    "phi" := "phi" + "w0c_6_12_1" * SIN(1 * 0.4 * "x") + "w0d_6_12_1" * COS(1 * 0.4 * "x");
    "phi" := "phi" + "w0c_6_12_2" * SIN(2 * 0.4 * "x") + "w0d_6_12_2" * COS(2 * 0.4 * "x");
    "phi" := "phi" + "w0c_6_12_3" * SIN(3 * 0.4 * "x") + "w0d_6_12_3" * COS(3 * 0.4 * "x");
    "phi" := "phi" + "w0c_6_12_4" * SIN(4 * 0.4 * "x") + "w0d_6_12_4" * COS(4 * 0.4 * "x");
    "phi" := "phi" + "w0c_6_12_5" * SIN(5 * 0.4 * "x") + "w0d_6_12_5" * COS(5 * 0.4 * "x");
    "phi" := "phi" + "w0c_6_12_6" * SIN(6 * 0.4 * "x") + "w0d_6_12_6" * COS(6 * 0.4 * "x");
    "acc" := "acc" + "phi";
    "x" := "feat_13";
    "phi" := "w0b_6_13" * "x" / (1.0 + EXP(-"x"));
    "phi" := "phi" + "w0c_6_13_1" * SIN(1 * 0.4 * "x") + "w0d_6_13_1" * COS(1 * 0.4 * "x");
    "phi" := "phi" + "w0c_6_13_2" * SIN(2 * 0.4 * "x") + "w0d_6_13_2" * COS(2 * 0.4 * "x");
    "phi" := "phi" + "w0c_6_13_3" * SIN(3 * 0.4 * "x") + "w0d_6_13_3" * COS(3 * 0.4 * "x");
    "phi" := "phi" + "w0c_6_13_4" * SIN(4 * 0.4 * "x") + "w0d_6_13_4" * COS(4 * 0.4 * "x");
    "phi" := "phi" + "w0c_6_13_5" * SIN(5 * 0.4 * "x") + "w0d_6_13_5" * COS(5 * 0.4 * "x");
    "phi" := "phi" + "w0c_6_13_6" * SIN(6 * 0.4 * "x") + "w0d_6_13_6" * COS(6 * 0.4 * "x");
    "acc" := "acc" + "phi";
    "x" := "feat_14";
    "phi" := "w0b_6_14" * "x" / (1.0 + EXP(-"x"));
    "phi" := "phi" + "w0c_6_14_1" * SIN(1 * 0.4 * "x") + "w0d_6_14_1" * COS(1 * 0.4 * "x");
    "phi" := "phi" + "w0c_6_14_2" * SIN(2 * 0.4 * "x") + "w0d_6_14_2" * COS(2 * 0.4 * "x");
    "phi" := "phi" + "w0c_6_14_3" * SIN(3 * 0.4 * "x") + "w0d_6_14_3" * COS(3 * 0.4 * "x");
    "phi" := "phi" + "w0c_6_14_4" * SIN(4 * 0.4 * "x") + "w0d_6_14_4" * COS(4 * 0.4 * "x");
    "phi" := "phi" + "w0c_6_14_5" * SIN(5 * 0.4 * "x") + "w0d_6_14_5" * COS(5 * 0.4 * "x");
    "phi" := "phi" + "w0c_6_14_6" * SIN(6 * 0.4 * "x") + "w0d_6_14_6" * COS(6 * 0.4 * "x");
    "acc" := "acc" + "phi";
    "x" := "feat_15";
    "phi" := "w0b_6_15" * "x" / (1.0 + EXP(-"x"));
    "phi" := "phi" + "w0c_6_15_1" * SIN(1 * 0.4 * "x") + "w0d_6_15_1" * COS(1 * 0.4 * "x");
    "phi" := "phi" + "w0c_6_15_2" * SIN(2 * 0.4 * "x") + "w0d_6_15_2" * COS(2 * 0.4 * "x");
    "phi" := "phi" + "w0c_6_15_3" * SIN(3 * 0.4 * "x") + "w0d_6_15_3" * COS(3 * 0.4 * "x");
    "phi" := "phi" + "w0c_6_15_4" * SIN(4 * 0.4 * "x") + "w0d_6_15_4" * COS(4 * 0.4 * "x");
    "phi" := "phi" + "w0c_6_15_5" * SIN(5 * 0.4 * "x") + "w0d_6_15_5" * COS(5 * 0.4 * "x");
    "phi" := "phi" + "w0c_6_15_6" * SIN(6 * 0.4 * "x") + "w0d_6_15_6" * COS(6 * 0.4 * "x");
    "acc" := "acc" + "phi";
    "x" := "feat_16";
    "phi" := "w0b_6_16" * "x" / (1.0 + EXP(-"x"));
    "phi" := "phi" + "w0c_6_16_1" * SIN(1 * 0.4 * "x") + "w0d_6_16_1" * COS(1 * 0.4 * "x");
    "phi" := "phi" + "w0c_6_16_2" * SIN(2 * 0.4 * "x") + "w0d_6_16_2" * COS(2 * 0.4 * "x");
    "phi" := "phi" + "w0c_6_16_3" * SIN(3 * 0.4 * "x") + "w0d_6_16_3" * COS(3 * 0.4 * "x");
    "phi" := "phi" + "w0c_6_16_4" * SIN(4 * 0.4 * "x") + "w0d_6_16_4" * COS(4 * 0.4 * "x");
    "phi" := "phi" + "w0c_6_16_5" * SIN(5 * 0.4 * "x") + "w0d_6_16_5" * COS(5 * 0.4 * "x");
    "phi" := "phi" + "w0c_6_16_6" * SIN(6 * 0.4 * "x") + "w0d_6_16_6" * COS(6 * 0.4 * "x");
    "acc" := "acc" + "phi";
    "x" := "feat_17";
    "phi" := "w0b_6_17" * "x" / (1.0 + EXP(-"x"));
    "phi" := "phi" + "w0c_6_17_1" * SIN(1 * 0.4 * "x") + "w0d_6_17_1" * COS(1 * 0.4 * "x");
    "phi" := "phi" + "w0c_6_17_2" * SIN(2 * 0.4 * "x") + "w0d_6_17_2" * COS(2 * 0.4 * "x");
    "phi" := "phi" + "w0c_6_17_3" * SIN(3 * 0.4 * "x") + "w0d_6_17_3" * COS(3 * 0.4 * "x");
    "phi" := "phi" + "w0c_6_17_4" * SIN(4 * 0.4 * "x") + "w0d_6_17_4" * COS(4 * 0.4 * "x");
    "phi" := "phi" + "w0c_6_17_5" * SIN(5 * 0.4 * "x") + "w0d_6_17_5" * COS(5 * 0.4 * "x");
    "phi" := "phi" + "w0c_6_17_6" * SIN(6 * 0.4 * "x") + "w0d_6_17_6" * COS(6 * 0.4 * "x");
    "acc" := "acc" + "phi";
    "x" := "feat_18";
    "phi" := "w0b_6_18" * "x" / (1.0 + EXP(-"x"));
    "phi" := "phi" + "w0c_6_18_1" * SIN(1 * 0.4 * "x") + "w0d_6_18_1" * COS(1 * 0.4 * "x");
    "phi" := "phi" + "w0c_6_18_2" * SIN(2 * 0.4 * "x") + "w0d_6_18_2" * COS(2 * 0.4 * "x");
    "phi" := "phi" + "w0c_6_18_3" * SIN(3 * 0.4 * "x") + "w0d_6_18_3" * COS(3 * 0.4 * "x");
    "phi" := "phi" + "w0c_6_18_4" * SIN(4 * 0.4 * "x") + "w0d_6_18_4" * COS(4 * 0.4 * "x");
    "phi" := "phi" + "w0c_6_18_5" * SIN(5 * 0.4 * "x") + "w0d_6_18_5" * COS(5 * 0.4 * "x");
    "phi" := "phi" + "w0c_6_18_6" * SIN(6 * 0.4 * "x") + "w0d_6_18_6" * COS(6 * 0.4 * "x");
    "acc" := "acc" + "phi";
    "x" := "feat_19";
    "phi" := "w0b_6_19" * "x" / (1.0 + EXP(-"x"));
    "phi" := "phi" + "w0c_6_19_1" * SIN(1 * 0.4 * "x") + "w0d_6_19_1" * COS(1 * 0.4 * "x");
    "phi" := "phi" + "w0c_6_19_2" * SIN(2 * 0.4 * "x") + "w0d_6_19_2" * COS(2 * 0.4 * "x");
    "phi" := "phi" + "w0c_6_19_3" * SIN(3 * 0.4 * "x") + "w0d_6_19_3" * COS(3 * 0.4 * "x");
    "phi" := "phi" + "w0c_6_19_4" * SIN(4 * 0.4 * "x") + "w0d_6_19_4" * COS(4 * 0.4 * "x");
    "phi" := "phi" + "w0c_6_19_5" * SIN(5 * 0.4 * "x") + "w0d_6_19_5" * COS(5 * 0.4 * "x");
    "phi" := "phi" + "w0c_6_19_6" * SIN(6 * 0.4 * "x") + "w0d_6_19_6" * COS(6 * 0.4 * "x");
    "acc" := "acc" + "phi";
    "x" := "feat_20";
    "phi" := "w0b_6_20" * "x" / (1.0 + EXP(-"x"));
    "phi" := "phi" + "w0c_6_20_1" * SIN(1 * 0.4 * "x") + "w0d_6_20_1" * COS(1 * 0.4 * "x");
    "phi" := "phi" + "w0c_6_20_2" * SIN(2 * 0.4 * "x") + "w0d_6_20_2" * COS(2 * 0.4 * "x");
    "phi" := "phi" + "w0c_6_20_3" * SIN(3 * 0.4 * "x") + "w0d_6_20_3" * COS(3 * 0.4 * "x");
    "phi" := "phi" + "w0c_6_20_4" * SIN(4 * 0.4 * "x") + "w0d_6_20_4" * COS(4 * 0.4 * "x");
    "phi" := "phi" + "w0c_6_20_5" * SIN(5 * 0.4 * "x") + "w0d_6_20_5" * COS(5 * 0.4 * "x");
    "phi" := "phi" + "w0c_6_20_6" * SIN(6 * 0.4 * "x") + "w0d_6_20_6" * COS(6 * 0.4 * "x");
    "acc" := "acc" + "phi";
    "x" := "feat_21";
    "phi" := "w0b_6_21" * "x" / (1.0 + EXP(-"x"));
    "phi" := "phi" + "w0c_6_21_1" * SIN(1 * 0.4 * "x") + "w0d_6_21_1" * COS(1 * 0.4 * "x");
    "phi" := "phi" + "w0c_6_21_2" * SIN(2 * 0.4 * "x") + "w0d_6_21_2" * COS(2 * 0.4 * "x");
    "phi" := "phi" + "w0c_6_21_3" * SIN(3 * 0.4 * "x") + "w0d_6_21_3" * COS(3 * 0.4 * "x");
    "phi" := "phi" + "w0c_6_21_4" * SIN(4 * 0.4 * "x") + "w0d_6_21_4" * COS(4 * 0.4 * "x");
    "phi" := "phi" + "w0c_6_21_5" * SIN(5 * 0.4 * "x") + "w0d_6_21_5" * COS(5 * 0.4 * "x");
    "phi" := "phi" + "w0c_6_21_6" * SIN(6 * 0.4 * "x") + "w0d_6_21_6" * COS(6 * 0.4 * "x");
    "acc" := "acc" + "phi";
    "x" := "feat_22";
    "phi" := "w0b_6_22" * "x" / (1.0 + EXP(-"x"));
    "phi" := "phi" + "w0c_6_22_1" * SIN(1 * 0.4 * "x") + "w0d_6_22_1" * COS(1 * 0.4 * "x");
    "phi" := "phi" + "w0c_6_22_2" * SIN(2 * 0.4 * "x") + "w0d_6_22_2" * COS(2 * 0.4 * "x");
    "phi" := "phi" + "w0c_6_22_3" * SIN(3 * 0.4 * "x") + "w0d_6_22_3" * COS(3 * 0.4 * "x");
    "phi" := "phi" + "w0c_6_22_4" * SIN(4 * 0.4 * "x") + "w0d_6_22_4" * COS(4 * 0.4 * "x");
    "phi" := "phi" + "w0c_6_22_5" * SIN(5 * 0.4 * "x") + "w0d_6_22_5" * COS(5 * 0.4 * "x");
    "phi" := "phi" + "w0c_6_22_6" * SIN(6 * 0.4 * "x") + "w0d_6_22_6" * COS(6 * 0.4 * "x");
    "acc" := "acc" + "phi";
    "x" := "feat_23";
    "phi" := "w0b_6_23" * "x" / (1.0 + EXP(-"x"));
    "phi" := "phi" + "w0c_6_23_1" * SIN(1 * 0.4 * "x") + "w0d_6_23_1" * COS(1 * 0.4 * "x");
    "phi" := "phi" + "w0c_6_23_2" * SIN(2 * 0.4 * "x") + "w0d_6_23_2" * COS(2 * 0.4 * "x");
    "phi" := "phi" + "w0c_6_23_3" * SIN(3 * 0.4 * "x") + "w0d_6_23_3" * COS(3 * 0.4 * "x");
    "phi" := "phi" + "w0c_6_23_4" * SIN(4 * 0.4 * "x") + "w0d_6_23_4" * COS(4 * 0.4 * "x");
    "phi" := "phi" + "w0c_6_23_5" * SIN(5 * 0.4 * "x") + "w0d_6_23_5" * COS(5 * 0.4 * "x");
    "phi" := "phi" + "w0c_6_23_6" * SIN(6 * 0.4 * "x") + "w0d_6_23_6" * COS(6 * 0.4 * "x");
    "acc" := "acc" + "phi";
    "x" := "feat_24";
    "phi" := "w0b_6_24" * "x" / (1.0 + EXP(-"x"));
    "phi" := "phi" + "w0c_6_24_1" * SIN(1 * 0.4 * "x") + "w0d_6_24_1" * COS(1 * 0.4 * "x");
    "phi" := "phi" + "w0c_6_24_2" * SIN(2 * 0.4 * "x") + "w0d_6_24_2" * COS(2 * 0.4 * "x");
    "phi" := "phi" + "w0c_6_24_3" * SIN(3 * 0.4 * "x") + "w0d_6_24_3" * COS(3 * 0.4 * "x");
    "phi" := "phi" + "w0c_6_24_4" * SIN(4 * 0.4 * "x") + "w0d_6_24_4" * COS(4 * 0.4 * "x");
    "phi" := "phi" + "w0c_6_24_5" * SIN(5 * 0.4 * "x") + "w0d_6_24_5" * COS(5 * 0.4 * "x");
    "phi" := "phi" + "w0c_6_24_6" * SIN(6 * 0.4 * "x") + "w0d_6_24_6" * COS(6 * 0.4 * "x");
    "acc" := "acc" + "phi";
    "x" := "feat_25";
    "phi" := "w0b_6_25" * "x" / (1.0 + EXP(-"x"));
    "phi" := "phi" + "w0c_6_25_1" * SIN(1 * 0.4 * "x") + "w0d_6_25_1" * COS(1 * 0.4 * "x");
    "phi" := "phi" + "w0c_6_25_2" * SIN(2 * 0.4 * "x") + "w0d_6_25_2" * COS(2 * 0.4 * "x");
    "phi" := "phi" + "w0c_6_25_3" * SIN(3 * 0.4 * "x") + "w0d_6_25_3" * COS(3 * 0.4 * "x");
    "phi" := "phi" + "w0c_6_25_4" * SIN(4 * 0.4 * "x") + "w0d_6_25_4" * COS(4 * 0.4 * "x");
    "phi" := "phi" + "w0c_6_25_5" * SIN(5 * 0.4 * "x") + "w0d_6_25_5" * COS(5 * 0.4 * "x");
    "phi" := "phi" + "w0c_6_25_6" * SIN(6 * 0.4 * "x") + "w0d_6_25_6" * COS(6 * 0.4 * "x");
    "acc" := "acc" + "phi";
    "x" := "feat_26";
    "phi" := "w0b_6_26" * "x" / (1.0 + EXP(-"x"));
    "phi" := "phi" + "w0c_6_26_1" * SIN(1 * 0.4 * "x") + "w0d_6_26_1" * COS(1 * 0.4 * "x");
    "phi" := "phi" + "w0c_6_26_2" * SIN(2 * 0.4 * "x") + "w0d_6_26_2" * COS(2 * 0.4 * "x");
    "phi" := "phi" + "w0c_6_26_3" * SIN(3 * 0.4 * "x") + "w0d_6_26_3" * COS(3 * 0.4 * "x");
    "phi" := "phi" + "w0c_6_26_4" * SIN(4 * 0.4 * "x") + "w0d_6_26_4" * COS(4 * 0.4 * "x");
    "phi" := "phi" + "w0c_6_26_5" * SIN(5 * 0.4 * "x") + "w0d_6_26_5" * COS(5 * 0.4 * "x");
    "phi" := "phi" + "w0c_6_26_6" * SIN(6 * 0.4 * "x") + "w0d_6_26_6" * COS(6 * 0.4 * "x");
    "acc" := "acc" + "phi";
    "x" := "feat_27";
    "phi" := "w0b_6_27" * "x" / (1.0 + EXP(-"x"));
    "phi" := "phi" + "w0c_6_27_1" * SIN(1 * 0.4 * "x") + "w0d_6_27_1" * COS(1 * 0.4 * "x");
    "phi" := "phi" + "w0c_6_27_2" * SIN(2 * 0.4 * "x") + "w0d_6_27_2" * COS(2 * 0.4 * "x");
    "phi" := "phi" + "w0c_6_27_3" * SIN(3 * 0.4 * "x") + "w0d_6_27_3" * COS(3 * 0.4 * "x");
    "phi" := "phi" + "w0c_6_27_4" * SIN(4 * 0.4 * "x") + "w0d_6_27_4" * COS(4 * 0.4 * "x");
    "phi" := "phi" + "w0c_6_27_5" * SIN(5 * 0.4 * "x") + "w0d_6_27_5" * COS(5 * 0.4 * "x");
    "phi" := "phi" + "w0c_6_27_6" * SIN(6 * 0.4 * "x") + "w0d_6_27_6" * COS(6 * 0.4 * "x");
    "acc" := "acc" + "phi";
    "x" := "feat_28";
    "phi" := "w0b_6_28" * "x" / (1.0 + EXP(-"x"));
    "phi" := "phi" + "w0c_6_28_1" * SIN(1 * 0.4 * "x") + "w0d_6_28_1" * COS(1 * 0.4 * "x");
    "phi" := "phi" + "w0c_6_28_2" * SIN(2 * 0.4 * "x") + "w0d_6_28_2" * COS(2 * 0.4 * "x");
    "phi" := "phi" + "w0c_6_28_3" * SIN(3 * 0.4 * "x") + "w0d_6_28_3" * COS(3 * 0.4 * "x");
    "phi" := "phi" + "w0c_6_28_4" * SIN(4 * 0.4 * "x") + "w0d_6_28_4" * COS(4 * 0.4 * "x");
    "phi" := "phi" + "w0c_6_28_5" * SIN(5 * 0.4 * "x") + "w0d_6_28_5" * COS(5 * 0.4 * "x");
    "phi" := "phi" + "w0c_6_28_6" * SIN(6 * 0.4 * "x") + "w0d_6_28_6" * COS(6 * 0.4 * "x");
    "acc" := "acc" + "phi";
    "h1_6" := "acc" + "b0_6";
    "acc" := 0.0;
    "x" := "feat_1";
    "phi" := "w0b_7_1" * "x" / (1.0 + EXP(-"x"));
    "phi" := "phi" + "w0c_7_1_1" * SIN(1 * 0.4 * "x") + "w0d_7_1_1" * COS(1 * 0.4 * "x");
    "phi" := "phi" + "w0c_7_1_2" * SIN(2 * 0.4 * "x") + "w0d_7_1_2" * COS(2 * 0.4 * "x");
    "phi" := "phi" + "w0c_7_1_3" * SIN(3 * 0.4 * "x") + "w0d_7_1_3" * COS(3 * 0.4 * "x");
    "phi" := "phi" + "w0c_7_1_4" * SIN(4 * 0.4 * "x") + "w0d_7_1_4" * COS(4 * 0.4 * "x");
    "phi" := "phi" + "w0c_7_1_5" * SIN(5 * 0.4 * "x") + "w0d_7_1_5" * COS(5 * 0.4 * "x");
    "phi" := "phi" + "w0c_7_1_6" * SIN(6 * 0.4 * "x") + "w0d_7_1_6" * COS(6 * 0.4 * "x");
    "acc" := "acc" + "phi";
    "x" := "feat_2";
    "phi" := "w0b_7_2" * "x" / (1.0 + EXP(-"x"));
    "phi" := "phi" + "w0c_7_2_1" * SIN(1 * 0.4 * "x") + "w0d_7_2_1" * COS(1 * 0.4 * "x");
    "phi" := "phi" + "w0c_7_2_2" * SIN(2 * 0.4 * "x") + "w0d_7_2_2" * COS(2 * 0.4 * "x");
    "phi" := "phi" + "w0c_7_2_3" * SIN(3 * 0.4 * "x") + "w0d_7_2_3" * COS(3 * 0.4 * "x");
    "phi" := "phi" + "w0c_7_2_4" * SIN(4 * 0.4 * "x") + "w0d_7_2_4" * COS(4 * 0.4 * "x");
    "phi" := "phi" + "w0c_7_2_5" * SIN(5 * 0.4 * "x") + "w0d_7_2_5" * COS(5 * 0.4 * "x");
    "phi" := "phi" + "w0c_7_2_6" * SIN(6 * 0.4 * "x") + "w0d_7_2_6" * COS(6 * 0.4 * "x");
    "acc" := "acc" + "phi";
    "x" := "feat_3";
    "phi" := "w0b_7_3" * "x" / (1.0 + EXP(-"x"));
    "phi" := "phi" + "w0c_7_3_1" * SIN(1 * 0.4 * "x") + "w0d_7_3_1" * COS(1 * 0.4 * "x");
    "phi" := "phi" + "w0c_7_3_2" * SIN(2 * 0.4 * "x") + "w0d_7_3_2" * COS(2 * 0.4 * "x");
    "phi" := "phi" + "w0c_7_3_3" * SIN(3 * 0.4 * "x") + "w0d_7_3_3" * COS(3 * 0.4 * "x");
    "phi" := "phi" + "w0c_7_3_4" * SIN(4 * 0.4 * "x") + "w0d_7_3_4" * COS(4 * 0.4 * "x");
    "phi" := "phi" + "w0c_7_3_5" * SIN(5 * 0.4 * "x") + "w0d_7_3_5" * COS(5 * 0.4 * "x");
    "phi" := "phi" + "w0c_7_3_6" * SIN(6 * 0.4 * "x") + "w0d_7_3_6" * COS(6 * 0.4 * "x");
    "acc" := "acc" + "phi";
    "x" := "feat_4";
    "phi" := "w0b_7_4" * "x" / (1.0 + EXP(-"x"));
    "phi" := "phi" + "w0c_7_4_1" * SIN(1 * 0.4 * "x") + "w0d_7_4_1" * COS(1 * 0.4 * "x");
    "phi" := "phi" + "w0c_7_4_2" * SIN(2 * 0.4 * "x") + "w0d_7_4_2" * COS(2 * 0.4 * "x");
    "phi" := "phi" + "w0c_7_4_3" * SIN(3 * 0.4 * "x") + "w0d_7_4_3" * COS(3 * 0.4 * "x");
    "phi" := "phi" + "w0c_7_4_4" * SIN(4 * 0.4 * "x") + "w0d_7_4_4" * COS(4 * 0.4 * "x");
    "phi" := "phi" + "w0c_7_4_5" * SIN(5 * 0.4 * "x") + "w0d_7_4_5" * COS(5 * 0.4 * "x");
    "phi" := "phi" + "w0c_7_4_6" * SIN(6 * 0.4 * "x") + "w0d_7_4_6" * COS(6 * 0.4 * "x");
    "acc" := "acc" + "phi";
    "x" := "feat_5";
    "phi" := "w0b_7_5" * "x" / (1.0 + EXP(-"x"));
    "phi" := "phi" + "w0c_7_5_1" * SIN(1 * 0.4 * "x") + "w0d_7_5_1" * COS(1 * 0.4 * "x");
    "phi" := "phi" + "w0c_7_5_2" * SIN(2 * 0.4 * "x") + "w0d_7_5_2" * COS(2 * 0.4 * "x");
    "phi" := "phi" + "w0c_7_5_3" * SIN(3 * 0.4 * "x") + "w0d_7_5_3" * COS(3 * 0.4 * "x");
    "phi" := "phi" + "w0c_7_5_4" * SIN(4 * 0.4 * "x") + "w0d_7_5_4" * COS(4 * 0.4 * "x");
    "phi" := "phi" + "w0c_7_5_5" * SIN(5 * 0.4 * "x") + "w0d_7_5_5" * COS(5 * 0.4 * "x");
    "phi" := "phi" + "w0c_7_5_6" * SIN(6 * 0.4 * "x") + "w0d_7_5_6" * COS(6 * 0.4 * "x");
    "acc" := "acc" + "phi";
    "x" := "feat_6";
    "phi" := "w0b_7_6" * "x" / (1.0 + EXP(-"x"));
    "phi" := "phi" + "w0c_7_6_1" * SIN(1 * 0.4 * "x") + "w0d_7_6_1" * COS(1 * 0.4 * "x");
    "phi" := "phi" + "w0c_7_6_2" * SIN(2 * 0.4 * "x") + "w0d_7_6_2" * COS(2 * 0.4 * "x");
    "phi" := "phi" + "w0c_7_6_3" * SIN(3 * 0.4 * "x") + "w0d_7_6_3" * COS(3 * 0.4 * "x");
    "phi" := "phi" + "w0c_7_6_4" * SIN(4 * 0.4 * "x") + "w0d_7_6_4" * COS(4 * 0.4 * "x");
    "phi" := "phi" + "w0c_7_6_5" * SIN(5 * 0.4 * "x") + "w0d_7_6_5" * COS(5 * 0.4 * "x");
    "phi" := "phi" + "w0c_7_6_6" * SIN(6 * 0.4 * "x") + "w0d_7_6_6" * COS(6 * 0.4 * "x");
    "acc" := "acc" + "phi";
    "x" := "feat_7";
    "phi" := "w0b_7_7" * "x" / (1.0 + EXP(-"x"));
    "phi" := "phi" + "w0c_7_7_1" * SIN(1 * 0.4 * "x") + "w0d_7_7_1" * COS(1 * 0.4 * "x");
    "phi" := "phi" + "w0c_7_7_2" * SIN(2 * 0.4 * "x") + "w0d_7_7_2" * COS(2 * 0.4 * "x");
    "phi" := "phi" + "w0c_7_7_3" * SIN(3 * 0.4 * "x") + "w0d_7_7_3" * COS(3 * 0.4 * "x");
    "phi" := "phi" + "w0c_7_7_4" * SIN(4 * 0.4 * "x") + "w0d_7_7_4" * COS(4 * 0.4 * "x");
    "phi" := "phi" + "w0c_7_7_5" * SIN(5 * 0.4 * "x") + "w0d_7_7_5" * COS(5 * 0.4 * "x");
    "phi" := "phi" + "w0c_7_7_6" * SIN(6 * 0.4 * "x") + "w0d_7_7_6" * COS(6 * 0.4 * "x");
    "acc" := "acc" + "phi";
    "x" := "feat_8";
    "phi" := "w0b_7_8" * "x" / (1.0 + EXP(-"x"));
    "phi" := "phi" + "w0c_7_8_1" * SIN(1 * 0.4 * "x") + "w0d_7_8_1" * COS(1 * 0.4 * "x");
    "phi" := "phi" + "w0c_7_8_2" * SIN(2 * 0.4 * "x") + "w0d_7_8_2" * COS(2 * 0.4 * "x");
    "phi" := "phi" + "w0c_7_8_3" * SIN(3 * 0.4 * "x") + "w0d_7_8_3" * COS(3 * 0.4 * "x");
    "phi" := "phi" + "w0c_7_8_4" * SIN(4 * 0.4 * "x") + "w0d_7_8_4" * COS(4 * 0.4 * "x");
    "phi" := "phi" + "w0c_7_8_5" * SIN(5 * 0.4 * "x") + "w0d_7_8_5" * COS(5 * 0.4 * "x");
    "phi" := "phi" + "w0c_7_8_6" * SIN(6 * 0.4 * "x") + "w0d_7_8_6" * COS(6 * 0.4 * "x");
    "acc" := "acc" + "phi";
    "x" := "feat_9";
    "phi" := "w0b_7_9" * "x" / (1.0 + EXP(-"x"));
    "phi" := "phi" + "w0c_7_9_1" * SIN(1 * 0.4 * "x") + "w0d_7_9_1" * COS(1 * 0.4 * "x");
    "phi" := "phi" + "w0c_7_9_2" * SIN(2 * 0.4 * "x") + "w0d_7_9_2" * COS(2 * 0.4 * "x");
    "phi" := "phi" + "w0c_7_9_3" * SIN(3 * 0.4 * "x") + "w0d_7_9_3" * COS(3 * 0.4 * "x");
    "phi" := "phi" + "w0c_7_9_4" * SIN(4 * 0.4 * "x") + "w0d_7_9_4" * COS(4 * 0.4 * "x");
    "phi" := "phi" + "w0c_7_9_5" * SIN(5 * 0.4 * "x") + "w0d_7_9_5" * COS(5 * 0.4 * "x");
    "phi" := "phi" + "w0c_7_9_6" * SIN(6 * 0.4 * "x") + "w0d_7_9_6" * COS(6 * 0.4 * "x");
    "acc" := "acc" + "phi";
    "x" := "feat_10";
    "phi" := "w0b_7_10" * "x" / (1.0 + EXP(-"x"));
    "phi" := "phi" + "w0c_7_10_1" * SIN(1 * 0.4 * "x") + "w0d_7_10_1" * COS(1 * 0.4 * "x");
    "phi" := "phi" + "w0c_7_10_2" * SIN(2 * 0.4 * "x") + "w0d_7_10_2" * COS(2 * 0.4 * "x");
    "phi" := "phi" + "w0c_7_10_3" * SIN(3 * 0.4 * "x") + "w0d_7_10_3" * COS(3 * 0.4 * "x");
    "phi" := "phi" + "w0c_7_10_4" * SIN(4 * 0.4 * "x") + "w0d_7_10_4" * COS(4 * 0.4 * "x");
    "phi" := "phi" + "w0c_7_10_5" * SIN(5 * 0.4 * "x") + "w0d_7_10_5" * COS(5 * 0.4 * "x");
    "phi" := "phi" + "w0c_7_10_6" * SIN(6 * 0.4 * "x") + "w0d_7_10_6" * COS(6 * 0.4 * "x");
    "acc" := "acc" + "phi";
    "x" := "feat_11";
    "phi" := "w0b_7_11" * "x" / (1.0 + EXP(-"x"));
    "phi" := "phi" + "w0c_7_11_1" * SIN(1 * 0.4 * "x") + "w0d_7_11_1" * COS(1 * 0.4 * "x");
    "phi" := "phi" + "w0c_7_11_2" * SIN(2 * 0.4 * "x") + "w0d_7_11_2" * COS(2 * 0.4 * "x");
    "phi" := "phi" + "w0c_7_11_3" * SIN(3 * 0.4 * "x") + "w0d_7_11_3" * COS(3 * 0.4 * "x");
    "phi" := "phi" + "w0c_7_11_4" * SIN(4 * 0.4 * "x") + "w0d_7_11_4" * COS(4 * 0.4 * "x");
    "phi" := "phi" + "w0c_7_11_5" * SIN(5 * 0.4 * "x") + "w0d_7_11_5" * COS(5 * 0.4 * "x");
    "phi" := "phi" + "w0c_7_11_6" * SIN(6 * 0.4 * "x") + "w0d_7_11_6" * COS(6 * 0.4 * "x");
    "acc" := "acc" + "phi";
    "x" := "feat_12";
    "phi" := "w0b_7_12" * "x" / (1.0 + EXP(-"x"));
    "phi" := "phi" + "w0c_7_12_1" * SIN(1 * 0.4 * "x") + "w0d_7_12_1" * COS(1 * 0.4 * "x");
    "phi" := "phi" + "w0c_7_12_2" * SIN(2 * 0.4 * "x") + "w0d_7_12_2" * COS(2 * 0.4 * "x");
    "phi" := "phi" + "w0c_7_12_3" * SIN(3 * 0.4 * "x") + "w0d_7_12_3" * COS(3 * 0.4 * "x");
    "phi" := "phi" + "w0c_7_12_4" * SIN(4 * 0.4 * "x") + "w0d_7_12_4" * COS(4 * 0.4 * "x");
    "phi" := "phi" + "w0c_7_12_5" * SIN(5 * 0.4 * "x") + "w0d_7_12_5" * COS(5 * 0.4 * "x");
    "phi" := "phi" + "w0c_7_12_6" * SIN(6 * 0.4 * "x") + "w0d_7_12_6" * COS(6 * 0.4 * "x");
    "acc" := "acc" + "phi";
    "x" := "feat_13";
    "phi" := "w0b_7_13" * "x" / (1.0 + EXP(-"x"));
    "phi" := "phi" + "w0c_7_13_1" * SIN(1 * 0.4 * "x") + "w0d_7_13_1" * COS(1 * 0.4 * "x");
    "phi" := "phi" + "w0c_7_13_2" * SIN(2 * 0.4 * "x") + "w0d_7_13_2" * COS(2 * 0.4 * "x");
    "phi" := "phi" + "w0c_7_13_3" * SIN(3 * 0.4 * "x") + "w0d_7_13_3" * COS(3 * 0.4 * "x");
    "phi" := "phi" + "w0c_7_13_4" * SIN(4 * 0.4 * "x") + "w0d_7_13_4" * COS(4 * 0.4 * "x");
    "phi" := "phi" + "w0c_7_13_5" * SIN(5 * 0.4 * "x") + "w0d_7_13_5" * COS(5 * 0.4 * "x");
    "phi" := "phi" + "w0c_7_13_6" * SIN(6 * 0.4 * "x") + "w0d_7_13_6" * COS(6 * 0.4 * "x");
    "acc" := "acc" + "phi";
    "x" := "feat_14";
    "phi" := "w0b_7_14" * "x" / (1.0 + EXP(-"x"));
    "phi" := "phi" + "w0c_7_14_1" * SIN(1 * 0.4 * "x") + "w0d_7_14_1" * COS(1 * 0.4 * "x");
    "phi" := "phi" + "w0c_7_14_2" * SIN(2 * 0.4 * "x") + "w0d_7_14_2" * COS(2 * 0.4 * "x");
    "phi" := "phi" + "w0c_7_14_3" * SIN(3 * 0.4 * "x") + "w0d_7_14_3" * COS(3 * 0.4 * "x");
    "phi" := "phi" + "w0c_7_14_4" * SIN(4 * 0.4 * "x") + "w0d_7_14_4" * COS(4 * 0.4 * "x");
    "phi" := "phi" + "w0c_7_14_5" * SIN(5 * 0.4 * "x") + "w0d_7_14_5" * COS(5 * 0.4 * "x");
    "phi" := "phi" + "w0c_7_14_6" * SIN(6 * 0.4 * "x") + "w0d_7_14_6" * COS(6 * 0.4 * "x");
    "acc" := "acc" + "phi";
    "x" := "feat_15";
    "phi" := "w0b_7_15" * "x" / (1.0 + EXP(-"x"));
    "phi" := "phi" + "w0c_7_15_1" * SIN(1 * 0.4 * "x") + "w0d_7_15_1" * COS(1 * 0.4 * "x");
    "phi" := "phi" + "w0c_7_15_2" * SIN(2 * 0.4 * "x") + "w0d_7_15_2" * COS(2 * 0.4 * "x");
    "phi" := "phi" + "w0c_7_15_3" * SIN(3 * 0.4 * "x") + "w0d_7_15_3" * COS(3 * 0.4 * "x");
    "phi" := "phi" + "w0c_7_15_4" * SIN(4 * 0.4 * "x") + "w0d_7_15_4" * COS(4 * 0.4 * "x");
    "phi" := "phi" + "w0c_7_15_5" * SIN(5 * 0.4 * "x") + "w0d_7_15_5" * COS(5 * 0.4 * "x");
    "phi" := "phi" + "w0c_7_15_6" * SIN(6 * 0.4 * "x") + "w0d_7_15_6" * COS(6 * 0.4 * "x");
    "acc" := "acc" + "phi";
    "x" := "feat_16";
    "phi" := "w0b_7_16" * "x" / (1.0 + EXP(-"x"));
    "phi" := "phi" + "w0c_7_16_1" * SIN(1 * 0.4 * "x") + "w0d_7_16_1" * COS(1 * 0.4 * "x");
    "phi" := "phi" + "w0c_7_16_2" * SIN(2 * 0.4 * "x") + "w0d_7_16_2" * COS(2 * 0.4 * "x");
    "phi" := "phi" + "w0c_7_16_3" * SIN(3 * 0.4 * "x") + "w0d_7_16_3" * COS(3 * 0.4 * "x");
    "phi" := "phi" + "w0c_7_16_4" * SIN(4 * 0.4 * "x") + "w0d_7_16_4" * COS(4 * 0.4 * "x");
    "phi" := "phi" + "w0c_7_16_5" * SIN(5 * 0.4 * "x") + "w0d_7_16_5" * COS(5 * 0.4 * "x");
    "phi" := "phi" + "w0c_7_16_6" * SIN(6 * 0.4 * "x") + "w0d_7_16_6" * COS(6 * 0.4 * "x");
    "acc" := "acc" + "phi";
    "x" := "feat_17";
    "phi" := "w0b_7_17" * "x" / (1.0 + EXP(-"x"));
    "phi" := "phi" + "w0c_7_17_1" * SIN(1 * 0.4 * "x") + "w0d_7_17_1" * COS(1 * 0.4 * "x");
    "phi" := "phi" + "w0c_7_17_2" * SIN(2 * 0.4 * "x") + "w0d_7_17_2" * COS(2 * 0.4 * "x");
    "phi" := "phi" + "w0c_7_17_3" * SIN(3 * 0.4 * "x") + "w0d_7_17_3" * COS(3 * 0.4 * "x");
    "phi" := "phi" + "w0c_7_17_4" * SIN(4 * 0.4 * "x") + "w0d_7_17_4" * COS(4 * 0.4 * "x");
    "phi" := "phi" + "w0c_7_17_5" * SIN(5 * 0.4 * "x") + "w0d_7_17_5" * COS(5 * 0.4 * "x");
    "phi" := "phi" + "w0c_7_17_6" * SIN(6 * 0.4 * "x") + "w0d_7_17_6" * COS(6 * 0.4 * "x");
    "acc" := "acc" + "phi";
    "x" := "feat_18";
    "phi" := "w0b_7_18" * "x" / (1.0 + EXP(-"x"));
    "phi" := "phi" + "w0c_7_18_1" * SIN(1 * 0.4 * "x") + "w0d_7_18_1" * COS(1 * 0.4 * "x");
    "phi" := "phi" + "w0c_7_18_2" * SIN(2 * 0.4 * "x") + "w0d_7_18_2" * COS(2 * 0.4 * "x");
    "phi" := "phi" + "w0c_7_18_3" * SIN(3 * 0.4 * "x") + "w0d_7_18_3" * COS(3 * 0.4 * "x");
    "phi" := "phi" + "w0c_7_18_4" * SIN(4 * 0.4 * "x") + "w0d_7_18_4" * COS(4 * 0.4 * "x");
    "phi" := "phi" + "w0c_7_18_5" * SIN(5 * 0.4 * "x") + "w0d_7_18_5" * COS(5 * 0.4 * "x");
    "phi" := "phi" + "w0c_7_18_6" * SIN(6 * 0.4 * "x") + "w0d_7_18_6" * COS(6 * 0.4 * "x");
    "acc" := "acc" + "phi";
    "x" := "feat_19";
    "phi" := "w0b_7_19" * "x" / (1.0 + EXP(-"x"));
    "phi" := "phi" + "w0c_7_19_1" * SIN(1 * 0.4 * "x") + "w0d_7_19_1" * COS(1 * 0.4 * "x");
    "phi" := "phi" + "w0c_7_19_2" * SIN(2 * 0.4 * "x") + "w0d_7_19_2" * COS(2 * 0.4 * "x");
    "phi" := "phi" + "w0c_7_19_3" * SIN(3 * 0.4 * "x") + "w0d_7_19_3" * COS(3 * 0.4 * "x");
    "phi" := "phi" + "w0c_7_19_4" * SIN(4 * 0.4 * "x") + "w0d_7_19_4" * COS(4 * 0.4 * "x");
    "phi" := "phi" + "w0c_7_19_5" * SIN(5 * 0.4 * "x") + "w0d_7_19_5" * COS(5 * 0.4 * "x");
    "phi" := "phi" + "w0c_7_19_6" * SIN(6 * 0.4 * "x") + "w0d_7_19_6" * COS(6 * 0.4 * "x");
    "acc" := "acc" + "phi";
    "x" := "feat_20";
    "phi" := "w0b_7_20" * "x" / (1.0 + EXP(-"x"));
    "phi" := "phi" + "w0c_7_20_1" * SIN(1 * 0.4 * "x") + "w0d_7_20_1" * COS(1 * 0.4 * "x");
    "phi" := "phi" + "w0c_7_20_2" * SIN(2 * 0.4 * "x") + "w0d_7_20_2" * COS(2 * 0.4 * "x");
    "phi" := "phi" + "w0c_7_20_3" * SIN(3 * 0.4 * "x") + "w0d_7_20_3" * COS(3 * 0.4 * "x");
    "phi" := "phi" + "w0c_7_20_4" * SIN(4 * 0.4 * "x") + "w0d_7_20_4" * COS(4 * 0.4 * "x");
    "phi" := "phi" + "w0c_7_20_5" * SIN(5 * 0.4 * "x") + "w0d_7_20_5" * COS(5 * 0.4 * "x");
    "phi" := "phi" + "w0c_7_20_6" * SIN(6 * 0.4 * "x") + "w0d_7_20_6" * COS(6 * 0.4 * "x");
    "acc" := "acc" + "phi";
    "x" := "feat_21";
    "phi" := "w0b_7_21" * "x" / (1.0 + EXP(-"x"));
    "phi" := "phi" + "w0c_7_21_1" * SIN(1 * 0.4 * "x") + "w0d_7_21_1" * COS(1 * 0.4 * "x");
    "phi" := "phi" + "w0c_7_21_2" * SIN(2 * 0.4 * "x") + "w0d_7_21_2" * COS(2 * 0.4 * "x");
    "phi" := "phi" + "w0c_7_21_3" * SIN(3 * 0.4 * "x") + "w0d_7_21_3" * COS(3 * 0.4 * "x");
    "phi" := "phi" + "w0c_7_21_4" * SIN(4 * 0.4 * "x") + "w0d_7_21_4" * COS(4 * 0.4 * "x");
    "phi" := "phi" + "w0c_7_21_5" * SIN(5 * 0.4 * "x") + "w0d_7_21_5" * COS(5 * 0.4 * "x");
    "phi" := "phi" + "w0c_7_21_6" * SIN(6 * 0.4 * "x") + "w0d_7_21_6" * COS(6 * 0.4 * "x");
    "acc" := "acc" + "phi";
    "x" := "feat_22";
    "phi" := "w0b_7_22" * "x" / (1.0 + EXP(-"x"));
    "phi" := "phi" + "w0c_7_22_1" * SIN(1 * 0.4 * "x") + "w0d_7_22_1" * COS(1 * 0.4 * "x");
    "phi" := "phi" + "w0c_7_22_2" * SIN(2 * 0.4 * "x") + "w0d_7_22_2" * COS(2 * 0.4 * "x");
    "phi" := "phi" + "w0c_7_22_3" * SIN(3 * 0.4 * "x") + "w0d_7_22_3" * COS(3 * 0.4 * "x");
    "phi" := "phi" + "w0c_7_22_4" * SIN(4 * 0.4 * "x") + "w0d_7_22_4" * COS(4 * 0.4 * "x");
    "phi" := "phi" + "w0c_7_22_5" * SIN(5 * 0.4 * "x") + "w0d_7_22_5" * COS(5 * 0.4 * "x");
    "phi" := "phi" + "w0c_7_22_6" * SIN(6 * 0.4 * "x") + "w0d_7_22_6" * COS(6 * 0.4 * "x");
    "acc" := "acc" + "phi";
    "x" := "feat_23";
    "phi" := "w0b_7_23" * "x" / (1.0 + EXP(-"x"));
    "phi" := "phi" + "w0c_7_23_1" * SIN(1 * 0.4 * "x") + "w0d_7_23_1" * COS(1 * 0.4 * "x");
    "phi" := "phi" + "w0c_7_23_2" * SIN(2 * 0.4 * "x") + "w0d_7_23_2" * COS(2 * 0.4 * "x");
    "phi" := "phi" + "w0c_7_23_3" * SIN(3 * 0.4 * "x") + "w0d_7_23_3" * COS(3 * 0.4 * "x");
    "phi" := "phi" + "w0c_7_23_4" * SIN(4 * 0.4 * "x") + "w0d_7_23_4" * COS(4 * 0.4 * "x");
    "phi" := "phi" + "w0c_7_23_5" * SIN(5 * 0.4 * "x") + "w0d_7_23_5" * COS(5 * 0.4 * "x");
    "phi" := "phi" + "w0c_7_23_6" * SIN(6 * 0.4 * "x") + "w0d_7_23_6" * COS(6 * 0.4 * "x");
    "acc" := "acc" + "phi";
    "x" := "feat_24";
    "phi" := "w0b_7_24" * "x" / (1.0 + EXP(-"x"));
    "phi" := "phi" + "w0c_7_24_1" * SIN(1 * 0.4 * "x") + "w0d_7_24_1" * COS(1 * 0.4 * "x");
    "phi" := "phi" + "w0c_7_24_2" * SIN(2 * 0.4 * "x") + "w0d_7_24_2" * COS(2 * 0.4 * "x");
    "phi" := "phi" + "w0c_7_24_3" * SIN(3 * 0.4 * "x") + "w0d_7_24_3" * COS(3 * 0.4 * "x");
    "phi" := "phi" + "w0c_7_24_4" * SIN(4 * 0.4 * "x") + "w0d_7_24_4" * COS(4 * 0.4 * "x");
    "phi" := "phi" + "w0c_7_24_5" * SIN(5 * 0.4 * "x") + "w0d_7_24_5" * COS(5 * 0.4 * "x");
    "phi" := "phi" + "w0c_7_24_6" * SIN(6 * 0.4 * "x") + "w0d_7_24_6" * COS(6 * 0.4 * "x");
    "acc" := "acc" + "phi";
    "x" := "feat_25";
    "phi" := "w0b_7_25" * "x" / (1.0 + EXP(-"x"));
    "phi" := "phi" + "w0c_7_25_1" * SIN(1 * 0.4 * "x") + "w0d_7_25_1" * COS(1 * 0.4 * "x");
    "phi" := "phi" + "w0c_7_25_2" * SIN(2 * 0.4 * "x") + "w0d_7_25_2" * COS(2 * 0.4 * "x");
    "phi" := "phi" + "w0c_7_25_3" * SIN(3 * 0.4 * "x") + "w0d_7_25_3" * COS(3 * 0.4 * "x");
    "phi" := "phi" + "w0c_7_25_4" * SIN(4 * 0.4 * "x") + "w0d_7_25_4" * COS(4 * 0.4 * "x");
    "phi" := "phi" + "w0c_7_25_5" * SIN(5 * 0.4 * "x") + "w0d_7_25_5" * COS(5 * 0.4 * "x");
    "phi" := "phi" + "w0c_7_25_6" * SIN(6 * 0.4 * "x") + "w0d_7_25_6" * COS(6 * 0.4 * "x");
    "acc" := "acc" + "phi";
    "x" := "feat_26";
    "phi" := "w0b_7_26" * "x" / (1.0 + EXP(-"x"));
    "phi" := "phi" + "w0c_7_26_1" * SIN(1 * 0.4 * "x") + "w0d_7_26_1" * COS(1 * 0.4 * "x");
    "phi" := "phi" + "w0c_7_26_2" * SIN(2 * 0.4 * "x") + "w0d_7_26_2" * COS(2 * 0.4 * "x");
    "phi" := "phi" + "w0c_7_26_3" * SIN(3 * 0.4 * "x") + "w0d_7_26_3" * COS(3 * 0.4 * "x");
    "phi" := "phi" + "w0c_7_26_4" * SIN(4 * 0.4 * "x") + "w0d_7_26_4" * COS(4 * 0.4 * "x");
    "phi" := "phi" + "w0c_7_26_5" * SIN(5 * 0.4 * "x") + "w0d_7_26_5" * COS(5 * 0.4 * "x");
    "phi" := "phi" + "w0c_7_26_6" * SIN(6 * 0.4 * "x") + "w0d_7_26_6" * COS(6 * 0.4 * "x");
    "acc" := "acc" + "phi";
    "x" := "feat_27";
    "phi" := "w0b_7_27" * "x" / (1.0 + EXP(-"x"));
    "phi" := "phi" + "w0c_7_27_1" * SIN(1 * 0.4 * "x") + "w0d_7_27_1" * COS(1 * 0.4 * "x");
    "phi" := "phi" + "w0c_7_27_2" * SIN(2 * 0.4 * "x") + "w0d_7_27_2" * COS(2 * 0.4 * "x");
    "phi" := "phi" + "w0c_7_27_3" * SIN(3 * 0.4 * "x") + "w0d_7_27_3" * COS(3 * 0.4 * "x");
    "phi" := "phi" + "w0c_7_27_4" * SIN(4 * 0.4 * "x") + "w0d_7_27_4" * COS(4 * 0.4 * "x");
    "phi" := "phi" + "w0c_7_27_5" * SIN(5 * 0.4 * "x") + "w0d_7_27_5" * COS(5 * 0.4 * "x");
    "phi" := "phi" + "w0c_7_27_6" * SIN(6 * 0.4 * "x") + "w0d_7_27_6" * COS(6 * 0.4 * "x");
    "acc" := "acc" + "phi";
    "x" := "feat_28";
    "phi" := "w0b_7_28" * "x" / (1.0 + EXP(-"x"));
    "phi" := "phi" + "w0c_7_28_1" * SIN(1 * 0.4 * "x") + "w0d_7_28_1" * COS(1 * 0.4 * "x");
    "phi" := "phi" + "w0c_7_28_2" * SIN(2 * 0.4 * "x") + "w0d_7_28_2" * COS(2 * 0.4 * "x");
    "phi" := "phi" + "w0c_7_28_3" * SIN(3 * 0.4 * "x") + "w0d_7_28_3" * COS(3 * 0.4 * "x");
    "phi" := "phi" + "w0c_7_28_4" * SIN(4 * 0.4 * "x") + "w0d_7_28_4" * COS(4 * 0.4 * "x");
    "phi" := "phi" + "w0c_7_28_5" * SIN(5 * 0.4 * "x") + "w0d_7_28_5" * COS(5 * 0.4 * "x");
    "phi" := "phi" + "w0c_7_28_6" * SIN(6 * 0.4 * "x") + "w0d_7_28_6" * COS(6 * 0.4 * "x");
    "acc" := "acc" + "phi";
    "h1_7" := "acc" + "b0_7";
    "acc" := 0.0;
    "x" := "feat_1";
    "phi" := "w0b_8_1" * "x" / (1.0 + EXP(-"x"));
    "phi" := "phi" + "w0c_8_1_1" * SIN(1 * 0.4 * "x") + "w0d_8_1_1" * COS(1 * 0.4 * "x");
    "phi" := "phi" + "w0c_8_1_2" * SIN(2 * 0.4 * "x") + "w0d_8_1_2" * COS(2 * 0.4 * "x");
    "phi" := "phi" + "w0c_8_1_3" * SIN(3 * 0.4 * "x") + "w0d_8_1_3" * COS(3 * 0.4 * "x");
    "phi" := "phi" + "w0c_8_1_4" * SIN(4 * 0.4 * "x") + "w0d_8_1_4" * COS(4 * 0.4 * "x");
    "phi" := "phi" + "w0c_8_1_5" * SIN(5 * 0.4 * "x") + "w0d_8_1_5" * COS(5 * 0.4 * "x");
    "phi" := "phi" + "w0c_8_1_6" * SIN(6 * 0.4 * "x") + "w0d_8_1_6" * COS(6 * 0.4 * "x");
    "acc" := "acc" + "phi";
    "x" := "feat_2";
    "phi" := "w0b_8_2" * "x" / (1.0 + EXP(-"x"));
    "phi" := "phi" + "w0c_8_2_1" * SIN(1 * 0.4 * "x") + "w0d_8_2_1" * COS(1 * 0.4 * "x");
    "phi" := "phi" + "w0c_8_2_2" * SIN(2 * 0.4 * "x") + "w0d_8_2_2" * COS(2 * 0.4 * "x");
    "phi" := "phi" + "w0c_8_2_3" * SIN(3 * 0.4 * "x") + "w0d_8_2_3" * COS(3 * 0.4 * "x");
    "phi" := "phi" + "w0c_8_2_4" * SIN(4 * 0.4 * "x") + "w0d_8_2_4" * COS(4 * 0.4 * "x");
    "phi" := "phi" + "w0c_8_2_5" * SIN(5 * 0.4 * "x") + "w0d_8_2_5" * COS(5 * 0.4 * "x");
    "phi" := "phi" + "w0c_8_2_6" * SIN(6 * 0.4 * "x") + "w0d_8_2_6" * COS(6 * 0.4 * "x");
    "acc" := "acc" + "phi";
    "x" := "feat_3";
    "phi" := "w0b_8_3" * "x" / (1.0 + EXP(-"x"));
    "phi" := "phi" + "w0c_8_3_1" * SIN(1 * 0.4 * "x") + "w0d_8_3_1" * COS(1 * 0.4 * "x");
    "phi" := "phi" + "w0c_8_3_2" * SIN(2 * 0.4 * "x") + "w0d_8_3_2" * COS(2 * 0.4 * "x");
    "phi" := "phi" + "w0c_8_3_3" * SIN(3 * 0.4 * "x") + "w0d_8_3_3" * COS(3 * 0.4 * "x");
    "phi" := "phi" + "w0c_8_3_4" * SIN(4 * 0.4 * "x") + "w0d_8_3_4" * COS(4 * 0.4 * "x");
    "phi" := "phi" + "w0c_8_3_5" * SIN(5 * 0.4 * "x") + "w0d_8_3_5" * COS(5 * 0.4 * "x");
    "phi" := "phi" + "w0c_8_3_6" * SIN(6 * 0.4 * "x") + "w0d_8_3_6" * COS(6 * 0.4 * "x");
    "acc" := "acc" + "phi";
    "x" := "feat_4";
    "phi" := "w0b_8_4" * "x" / (1.0 + EXP(-"x"));
    "phi" := "phi" + "w0c_8_4_1" * SIN(1 * 0.4 * "x") + "w0d_8_4_1" * COS(1 * 0.4 * "x");
    "phi" := "phi" + "w0c_8_4_2" * SIN(2 * 0.4 * "x") + "w0d_8_4_2" * COS(2 * 0.4 * "x");
    "phi" := "phi" + "w0c_8_4_3" * SIN(3 * 0.4 * "x") + "w0d_8_4_3" * COS(3 * 0.4 * "x");
    "phi" := "phi" + "w0c_8_4_4" * SIN(4 * 0.4 * "x") + "w0d_8_4_4" * COS(4 * 0.4 * "x");
    "phi" := "phi" + "w0c_8_4_5" * SIN(5 * 0.4 * "x") + "w0d_8_4_5" * COS(5 * 0.4 * "x");
    "phi" := "phi" + "w0c_8_4_6" * SIN(6 * 0.4 * "x") + "w0d_8_4_6" * COS(6 * 0.4 * "x");
    "acc" := "acc" + "phi";
    "x" := "feat_5";
    "phi" := "w0b_8_5" * "x" / (1.0 + EXP(-"x"));
    "phi" := "phi" + "w0c_8_5_1" * SIN(1 * 0.4 * "x") + "w0d_8_5_1" * COS(1 * 0.4 * "x");
    "phi" := "phi" + "w0c_8_5_2" * SIN(2 * 0.4 * "x") + "w0d_8_5_2" * COS(2 * 0.4 * "x");
    "phi" := "phi" + "w0c_8_5_3" * SIN(3 * 0.4 * "x") + "w0d_8_5_3" * COS(3 * 0.4 * "x");
    "phi" := "phi" + "w0c_8_5_4" * SIN(4 * 0.4 * "x") + "w0d_8_5_4" * COS(4 * 0.4 * "x");
    "phi" := "phi" + "w0c_8_5_5" * SIN(5 * 0.4 * "x") + "w0d_8_5_5" * COS(5 * 0.4 * "x");
    "phi" := "phi" + "w0c_8_5_6" * SIN(6 * 0.4 * "x") + "w0d_8_5_6" * COS(6 * 0.4 * "x");
    "acc" := "acc" + "phi";
    "x" := "feat_6";
    "phi" := "w0b_8_6" * "x" / (1.0 + EXP(-"x"));
    "phi" := "phi" + "w0c_8_6_1" * SIN(1 * 0.4 * "x") + "w0d_8_6_1" * COS(1 * 0.4 * "x");
    "phi" := "phi" + "w0c_8_6_2" * SIN(2 * 0.4 * "x") + "w0d_8_6_2" * COS(2 * 0.4 * "x");
    "phi" := "phi" + "w0c_8_6_3" * SIN(3 * 0.4 * "x") + "w0d_8_6_3" * COS(3 * 0.4 * "x");
    "phi" := "phi" + "w0c_8_6_4" * SIN(4 * 0.4 * "x") + "w0d_8_6_4" * COS(4 * 0.4 * "x");
    "phi" := "phi" + "w0c_8_6_5" * SIN(5 * 0.4 * "x") + "w0d_8_6_5" * COS(5 * 0.4 * "x");
    "phi" := "phi" + "w0c_8_6_6" * SIN(6 * 0.4 * "x") + "w0d_8_6_6" * COS(6 * 0.4 * "x");
    "acc" := "acc" + "phi";
    "x" := "feat_7";
    "phi" := "w0b_8_7" * "x" / (1.0 + EXP(-"x"));
    "phi" := "phi" + "w0c_8_7_1" * SIN(1 * 0.4 * "x") + "w0d_8_7_1" * COS(1 * 0.4 * "x");
    "phi" := "phi" + "w0c_8_7_2" * SIN(2 * 0.4 * "x") + "w0d_8_7_2" * COS(2 * 0.4 * "x");
    "phi" := "phi" + "w0c_8_7_3" * SIN(3 * 0.4 * "x") + "w0d_8_7_3" * COS(3 * 0.4 * "x");
    "phi" := "phi" + "w0c_8_7_4" * SIN(4 * 0.4 * "x") + "w0d_8_7_4" * COS(4 * 0.4 * "x");
    "phi" := "phi" + "w0c_8_7_5" * SIN(5 * 0.4 * "x") + "w0d_8_7_5" * COS(5 * 0.4 * "x");
    "phi" := "phi" + "w0c_8_7_6" * SIN(6 * 0.4 * "x") + "w0d_8_7_6" * COS(6 * 0.4 * "x");
    "acc" := "acc" + "phi";
    "x" := "feat_8";
    "phi" := "w0b_8_8" * "x" / (1.0 + EXP(-"x"));
    "phi" := "phi" + "w0c_8_8_1" * SIN(1 * 0.4 * "x") + "w0d_8_8_1" * COS(1 * 0.4 * "x");
    "phi" := "phi" + "w0c_8_8_2" * SIN(2 * 0.4 * "x") + "w0d_8_8_2" * COS(2 * 0.4 * "x");
    "phi" := "phi" + "w0c_8_8_3" * SIN(3 * 0.4 * "x") + "w0d_8_8_3" * COS(3 * 0.4 * "x");
    "phi" := "phi" + "w0c_8_8_4" * SIN(4 * 0.4 * "x") + "w0d_8_8_4" * COS(4 * 0.4 * "x");
    "phi" := "phi" + "w0c_8_8_5" * SIN(5 * 0.4 * "x") + "w0d_8_8_5" * COS(5 * 0.4 * "x");
    "phi" := "phi" + "w0c_8_8_6" * SIN(6 * 0.4 * "x") + "w0d_8_8_6" * COS(6 * 0.4 * "x");
    "acc" := "acc" + "phi";
    "x" := "feat_9";
    "phi" := "w0b_8_9" * "x" / (1.0 + EXP(-"x"));
    "phi" := "phi" + "w0c_8_9_1" * SIN(1 * 0.4 * "x") + "w0d_8_9_1" * COS(1 * 0.4 * "x");
    "phi" := "phi" + "w0c_8_9_2" * SIN(2 * 0.4 * "x") + "w0d_8_9_2" * COS(2 * 0.4 * "x");
    "phi" := "phi" + "w0c_8_9_3" * SIN(3 * 0.4 * "x") + "w0d_8_9_3" * COS(3 * 0.4 * "x");
    "phi" := "phi" + "w0c_8_9_4" * SIN(4 * 0.4 * "x") + "w0d_8_9_4" * COS(4 * 0.4 * "x");
    "phi" := "phi" + "w0c_8_9_5" * SIN(5 * 0.4 * "x") + "w0d_8_9_5" * COS(5 * 0.4 * "x");
    "phi" := "phi" + "w0c_8_9_6" * SIN(6 * 0.4 * "x") + "w0d_8_9_6" * COS(6 * 0.4 * "x");
    "acc" := "acc" + "phi";
    "x" := "feat_10";
    "phi" := "w0b_8_10" * "x" / (1.0 + EXP(-"x"));
    "phi" := "phi" + "w0c_8_10_1" * SIN(1 * 0.4 * "x") + "w0d_8_10_1" * COS(1 * 0.4 * "x");
    "phi" := "phi" + "w0c_8_10_2" * SIN(2 * 0.4 * "x") + "w0d_8_10_2" * COS(2 * 0.4 * "x");
    "phi" := "phi" + "w0c_8_10_3" * SIN(3 * 0.4 * "x") + "w0d_8_10_3" * COS(3 * 0.4 * "x");
    "phi" := "phi" + "w0c_8_10_4" * SIN(4 * 0.4 * "x") + "w0d_8_10_4" * COS(4 * 0.4 * "x");
    "phi" := "phi" + "w0c_8_10_5" * SIN(5 * 0.4 * "x") + "w0d_8_10_5" * COS(5 * 0.4 * "x");
    "phi" := "phi" + "w0c_8_10_6" * SIN(6 * 0.4 * "x") + "w0d_8_10_6" * COS(6 * 0.4 * "x");
    "acc" := "acc" + "phi";
    "x" := "feat_11";
    "phi" := "w0b_8_11" * "x" / (1.0 + EXP(-"x"));
    "phi" := "phi" + "w0c_8_11_1" * SIN(1 * 0.4 * "x") + "w0d_8_11_1" * COS(1 * 0.4 * "x");
    "phi" := "phi" + "w0c_8_11_2" * SIN(2 * 0.4 * "x") + "w0d_8_11_2" * COS(2 * 0.4 * "x");
    "phi" := "phi" + "w0c_8_11_3" * SIN(3 * 0.4 * "x") + "w0d_8_11_3" * COS(3 * 0.4 * "x");
    "phi" := "phi" + "w0c_8_11_4" * SIN(4 * 0.4 * "x") + "w0d_8_11_4" * COS(4 * 0.4 * "x");
    "phi" := "phi" + "w0c_8_11_5" * SIN(5 * 0.4 * "x") + "w0d_8_11_5" * COS(5 * 0.4 * "x");
    "phi" := "phi" + "w0c_8_11_6" * SIN(6 * 0.4 * "x") + "w0d_8_11_6" * COS(6 * 0.4 * "x");
    "acc" := "acc" + "phi";
    "x" := "feat_12";
    "phi" := "w0b_8_12" * "x" / (1.0 + EXP(-"x"));
    "phi" := "phi" + "w0c_8_12_1" * SIN(1 * 0.4 * "x") + "w0d_8_12_1" * COS(1 * 0.4 * "x");
    "phi" := "phi" + "w0c_8_12_2" * SIN(2 * 0.4 * "x") + "w0d_8_12_2" * COS(2 * 0.4 * "x");
    "phi" := "phi" + "w0c_8_12_3" * SIN(3 * 0.4 * "x") + "w0d_8_12_3" * COS(3 * 0.4 * "x");
    "phi" := "phi" + "w0c_8_12_4" * SIN(4 * 0.4 * "x") + "w0d_8_12_4" * COS(4 * 0.4 * "x");
    "phi" := "phi" + "w0c_8_12_5" * SIN(5 * 0.4 * "x") + "w0d_8_12_5" * COS(5 * 0.4 * "x");
    "phi" := "phi" + "w0c_8_12_6" * SIN(6 * 0.4 * "x") + "w0d_8_12_6" * COS(6 * 0.4 * "x");
    "acc" := "acc" + "phi";
    "x" := "feat_13";
    "phi" := "w0b_8_13" * "x" / (1.0 + EXP(-"x"));
    "phi" := "phi" + "w0c_8_13_1" * SIN(1 * 0.4 * "x") + "w0d_8_13_1" * COS(1 * 0.4 * "x");
    "phi" := "phi" + "w0c_8_13_2" * SIN(2 * 0.4 * "x") + "w0d_8_13_2" * COS(2 * 0.4 * "x");
    "phi" := "phi" + "w0c_8_13_3" * SIN(3 * 0.4 * "x") + "w0d_8_13_3" * COS(3 * 0.4 * "x");
    "phi" := "phi" + "w0c_8_13_4" * SIN(4 * 0.4 * "x") + "w0d_8_13_4" * COS(4 * 0.4 * "x");
    "phi" := "phi" + "w0c_8_13_5" * SIN(5 * 0.4 * "x") + "w0d_8_13_5" * COS(5 * 0.4 * "x");
    "phi" := "phi" + "w0c_8_13_6" * SIN(6 * 0.4 * "x") + "w0d_8_13_6" * COS(6 * 0.4 * "x");
    "acc" := "acc" + "phi";
    "x" := "feat_14";
    "phi" := "w0b_8_14" * "x" / (1.0 + EXP(-"x"));
    "phi" := "phi" + "w0c_8_14_1" * SIN(1 * 0.4 * "x") + "w0d_8_14_1" * COS(1 * 0.4 * "x");
    "phi" := "phi" + "w0c_8_14_2" * SIN(2 * 0.4 * "x") + "w0d_8_14_2" * COS(2 * 0.4 * "x");
    "phi" := "phi" + "w0c_8_14_3" * SIN(3 * 0.4 * "x") + "w0d_8_14_3" * COS(3 * 0.4 * "x");
    "phi" := "phi" + "w0c_8_14_4" * SIN(4 * 0.4 * "x") + "w0d_8_14_4" * COS(4 * 0.4 * "x");
    "phi" := "phi" + "w0c_8_14_5" * SIN(5 * 0.4 * "x") + "w0d_8_14_5" * COS(5 * 0.4 * "x");
    "phi" := "phi" + "w0c_8_14_6" * SIN(6 * 0.4 * "x") + "w0d_8_14_6" * COS(6 * 0.4 * "x");
    "acc" := "acc" + "phi";
    "x" := "feat_15";
    "phi" := "w0b_8_15" * "x" / (1.0 + EXP(-"x"));
    "phi" := "phi" + "w0c_8_15_1" * SIN(1 * 0.4 * "x") + "w0d_8_15_1" * COS(1 * 0.4 * "x");
    "phi" := "phi" + "w0c_8_15_2" * SIN(2 * 0.4 * "x") + "w0d_8_15_2" * COS(2 * 0.4 * "x");
    "phi" := "phi" + "w0c_8_15_3" * SIN(3 * 0.4 * "x") + "w0d_8_15_3" * COS(3 * 0.4 * "x");
    "phi" := "phi" + "w0c_8_15_4" * SIN(4 * 0.4 * "x") + "w0d_8_15_4" * COS(4 * 0.4 * "x");
    "phi" := "phi" + "w0c_8_15_5" * SIN(5 * 0.4 * "x") + "w0d_8_15_5" * COS(5 * 0.4 * "x");
    "phi" := "phi" + "w0c_8_15_6" * SIN(6 * 0.4 * "x") + "w0d_8_15_6" * COS(6 * 0.4 * "x");
    "acc" := "acc" + "phi";
    "x" := "feat_16";
    "phi" := "w0b_8_16" * "x" / (1.0 + EXP(-"x"));
    "phi" := "phi" + "w0c_8_16_1" * SIN(1 * 0.4 * "x") + "w0d_8_16_1" * COS(1 * 0.4 * "x");
    "phi" := "phi" + "w0c_8_16_2" * SIN(2 * 0.4 * "x") + "w0d_8_16_2" * COS(2 * 0.4 * "x");
    "phi" := "phi" + "w0c_8_16_3" * SIN(3 * 0.4 * "x") + "w0d_8_16_3" * COS(3 * 0.4 * "x");
    "phi" := "phi" + "w0c_8_16_4" * SIN(4 * 0.4 * "x") + "w0d_8_16_4" * COS(4 * 0.4 * "x");
    "phi" := "phi" + "w0c_8_16_5" * SIN(5 * 0.4 * "x") + "w0d_8_16_5" * COS(5 * 0.4 * "x");
    "phi" := "phi" + "w0c_8_16_6" * SIN(6 * 0.4 * "x") + "w0d_8_16_6" * COS(6 * 0.4 * "x");
    "acc" := "acc" + "phi";
    "x" := "feat_17";
    "phi" := "w0b_8_17" * "x" / (1.0 + EXP(-"x"));
    "phi" := "phi" + "w0c_8_17_1" * SIN(1 * 0.4 * "x") + "w0d_8_17_1" * COS(1 * 0.4 * "x");
    "phi" := "phi" + "w0c_8_17_2" * SIN(2 * 0.4 * "x") + "w0d_8_17_2" * COS(2 * 0.4 * "x");
    "phi" := "phi" + "w0c_8_17_3" * SIN(3 * 0.4 * "x") + "w0d_8_17_3" * COS(3 * 0.4 * "x");
    "phi" := "phi" + "w0c_8_17_4" * SIN(4 * 0.4 * "x") + "w0d_8_17_4" * COS(4 * 0.4 * "x");
    "phi" := "phi" + "w0c_8_17_5" * SIN(5 * 0.4 * "x") + "w0d_8_17_5" * COS(5 * 0.4 * "x");
    "phi" := "phi" + "w0c_8_17_6" * SIN(6 * 0.4 * "x") + "w0d_8_17_6" * COS(6 * 0.4 * "x");
    "acc" := "acc" + "phi";
    "x" := "feat_18";
    "phi" := "w0b_8_18" * "x" / (1.0 + EXP(-"x"));
    "phi" := "phi" + "w0c_8_18_1" * SIN(1 * 0.4 * "x") + "w0d_8_18_1" * COS(1 * 0.4 * "x");
    "phi" := "phi" + "w0c_8_18_2" * SIN(2 * 0.4 * "x") + "w0d_8_18_2" * COS(2 * 0.4 * "x");
    "phi" := "phi" + "w0c_8_18_3" * SIN(3 * 0.4 * "x") + "w0d_8_18_3" * COS(3 * 0.4 * "x");
    "phi" := "phi" + "w0c_8_18_4" * SIN(4 * 0.4 * "x") + "w0d_8_18_4" * COS(4 * 0.4 * "x");
    "phi" := "phi" + "w0c_8_18_5" * SIN(5 * 0.4 * "x") + "w0d_8_18_5" * COS(5 * 0.4 * "x");
    "phi" := "phi" + "w0c_8_18_6" * SIN(6 * 0.4 * "x") + "w0d_8_18_6" * COS(6 * 0.4 * "x");
    "acc" := "acc" + "phi";
    "x" := "feat_19";
    "phi" := "w0b_8_19" * "x" / (1.0 + EXP(-"x"));
    "phi" := "phi" + "w0c_8_19_1" * SIN(1 * 0.4 * "x") + "w0d_8_19_1" * COS(1 * 0.4 * "x");
    "phi" := "phi" + "w0c_8_19_2" * SIN(2 * 0.4 * "x") + "w0d_8_19_2" * COS(2 * 0.4 * "x");
    "phi" := "phi" + "w0c_8_19_3" * SIN(3 * 0.4 * "x") + "w0d_8_19_3" * COS(3 * 0.4 * "x");
    "phi" := "phi" + "w0c_8_19_4" * SIN(4 * 0.4 * "x") + "w0d_8_19_4" * COS(4 * 0.4 * "x");
    "phi" := "phi" + "w0c_8_19_5" * SIN(5 * 0.4 * "x") + "w0d_8_19_5" * COS(5 * 0.4 * "x");
    "phi" := "phi" + "w0c_8_19_6" * SIN(6 * 0.4 * "x") + "w0d_8_19_6" * COS(6 * 0.4 * "x");
    "acc" := "acc" + "phi";
    "x" := "feat_20";
    "phi" := "w0b_8_20" * "x" / (1.0 + EXP(-"x"));
    "phi" := "phi" + "w0c_8_20_1" * SIN(1 * 0.4 * "x") + "w0d_8_20_1" * COS(1 * 0.4 * "x");
    "phi" := "phi" + "w0c_8_20_2" * SIN(2 * 0.4 * "x") + "w0d_8_20_2" * COS(2 * 0.4 * "x");
    "phi" := "phi" + "w0c_8_20_3" * SIN(3 * 0.4 * "x") + "w0d_8_20_3" * COS(3 * 0.4 * "x");
    "phi" := "phi" + "w0c_8_20_4" * SIN(4 * 0.4 * "x") + "w0d_8_20_4" * COS(4 * 0.4 * "x");
    "phi" := "phi" + "w0c_8_20_5" * SIN(5 * 0.4 * "x") + "w0d_8_20_5" * COS(5 * 0.4 * "x");
    "phi" := "phi" + "w0c_8_20_6" * SIN(6 * 0.4 * "x") + "w0d_8_20_6" * COS(6 * 0.4 * "x");
    "acc" := "acc" + "phi";
    "x" := "feat_21";
    "phi" := "w0b_8_21" * "x" / (1.0 + EXP(-"x"));
    "phi" := "phi" + "w0c_8_21_1" * SIN(1 * 0.4 * "x") + "w0d_8_21_1" * COS(1 * 0.4 * "x");
    "phi" := "phi" + "w0c_8_21_2" * SIN(2 * 0.4 * "x") + "w0d_8_21_2" * COS(2 * 0.4 * "x");
    "phi" := "phi" + "w0c_8_21_3" * SIN(3 * 0.4 * "x") + "w0d_8_21_3" * COS(3 * 0.4 * "x");
    "phi" := "phi" + "w0c_8_21_4" * SIN(4 * 0.4 * "x") + "w0d_8_21_4" * COS(4 * 0.4 * "x");
    "phi" := "phi" + "w0c_8_21_5" * SIN(5 * 0.4 * "x") + "w0d_8_21_5" * COS(5 * 0.4 * "x");
    "phi" := "phi" + "w0c_8_21_6" * SIN(6 * 0.4 * "x") + "w0d_8_21_6" * COS(6 * 0.4 * "x");
    "acc" := "acc" + "phi";
    "x" := "feat_22";
    "phi" := "w0b_8_22" * "x" / (1.0 + EXP(-"x"));
    "phi" := "phi" + "w0c_8_22_1" * SIN(1 * 0.4 * "x") + "w0d_8_22_1" * COS(1 * 0.4 * "x");
    "phi" := "phi" + "w0c_8_22_2" * SIN(2 * 0.4 * "x") + "w0d_8_22_2" * COS(2 * 0.4 * "x");
    "phi" := "phi" + "w0c_8_22_3" * SIN(3 * 0.4 * "x") + "w0d_8_22_3" * COS(3 * 0.4 * "x");
    "phi" := "phi" + "w0c_8_22_4" * SIN(4 * 0.4 * "x") + "w0d_8_22_4" * COS(4 * 0.4 * "x");
    "phi" := "phi" + "w0c_8_22_5" * SIN(5 * 0.4 * "x") + "w0d_8_22_5" * COS(5 * 0.4 * "x");
    "phi" := "phi" + "w0c_8_22_6" * SIN(6 * 0.4 * "x") + "w0d_8_22_6" * COS(6 * 0.4 * "x");
    "acc" := "acc" + "phi";
    "x" := "feat_23";
    "phi" := "w0b_8_23" * "x" / (1.0 + EXP(-"x"));
    "phi" := "phi" + "w0c_8_23_1" * SIN(1 * 0.4 * "x") + "w0d_8_23_1" * COS(1 * 0.4 * "x");
    "phi" := "phi" + "w0c_8_23_2" * SIN(2 * 0.4 * "x") + "w0d_8_23_2" * COS(2 * 0.4 * "x");
    "phi" := "phi" + "w0c_8_23_3" * SIN(3 * 0.4 * "x") + "w0d_8_23_3" * COS(3 * 0.4 * "x");
    "phi" := "phi" + "w0c_8_23_4" * SIN(4 * 0.4 * "x") + "w0d_8_23_4" * COS(4 * 0.4 * "x");
    "phi" := "phi" + "w0c_8_23_5" * SIN(5 * 0.4 * "x") + "w0d_8_23_5" * COS(5 * 0.4 * "x");
    "phi" := "phi" + "w0c_8_23_6" * SIN(6 * 0.4 * "x") + "w0d_8_23_6" * COS(6 * 0.4 * "x");
    "acc" := "acc" + "phi";
    "x" := "feat_24";
    "phi" := "w0b_8_24" * "x" / (1.0 + EXP(-"x"));
    "phi" := "phi" + "w0c_8_24_1" * SIN(1 * 0.4 * "x") + "w0d_8_24_1" * COS(1 * 0.4 * "x");
    "phi" := "phi" + "w0c_8_24_2" * SIN(2 * 0.4 * "x") + "w0d_8_24_2" * COS(2 * 0.4 * "x");
    "phi" := "phi" + "w0c_8_24_3" * SIN(3 * 0.4 * "x") + "w0d_8_24_3" * COS(3 * 0.4 * "x");
    "phi" := "phi" + "w0c_8_24_4" * SIN(4 * 0.4 * "x") + "w0d_8_24_4" * COS(4 * 0.4 * "x");
    "phi" := "phi" + "w0c_8_24_5" * SIN(5 * 0.4 * "x") + "w0d_8_24_5" * COS(5 * 0.4 * "x");
    "phi" := "phi" + "w0c_8_24_6" * SIN(6 * 0.4 * "x") + "w0d_8_24_6" * COS(6 * 0.4 * "x");
    "acc" := "acc" + "phi";
    "x" := "feat_25";
    "phi" := "w0b_8_25" * "x" / (1.0 + EXP(-"x"));
    "phi" := "phi" + "w0c_8_25_1" * SIN(1 * 0.4 * "x") + "w0d_8_25_1" * COS(1 * 0.4 * "x");
    "phi" := "phi" + "w0c_8_25_2" * SIN(2 * 0.4 * "x") + "w0d_8_25_2" * COS(2 * 0.4 * "x");
    "phi" := "phi" + "w0c_8_25_3" * SIN(3 * 0.4 * "x") + "w0d_8_25_3" * COS(3 * 0.4 * "x");
    "phi" := "phi" + "w0c_8_25_4" * SIN(4 * 0.4 * "x") + "w0d_8_25_4" * COS(4 * 0.4 * "x");
    "phi" := "phi" + "w0c_8_25_5" * SIN(5 * 0.4 * "x") + "w0d_8_25_5" * COS(5 * 0.4 * "x");
    "phi" := "phi" + "w0c_8_25_6" * SIN(6 * 0.4 * "x") + "w0d_8_25_6" * COS(6 * 0.4 * "x");
    "acc" := "acc" + "phi";
    "x" := "feat_26";
    "phi" := "w0b_8_26" * "x" / (1.0 + EXP(-"x"));
    "phi" := "phi" + "w0c_8_26_1" * SIN(1 * 0.4 * "x") + "w0d_8_26_1" * COS(1 * 0.4 * "x");
    "phi" := "phi" + "w0c_8_26_2" * SIN(2 * 0.4 * "x") + "w0d_8_26_2" * COS(2 * 0.4 * "x");
    "phi" := "phi" + "w0c_8_26_3" * SIN(3 * 0.4 * "x") + "w0d_8_26_3" * COS(3 * 0.4 * "x");
    "phi" := "phi" + "w0c_8_26_4" * SIN(4 * 0.4 * "x") + "w0d_8_26_4" * COS(4 * 0.4 * "x");
    "phi" := "phi" + "w0c_8_26_5" * SIN(5 * 0.4 * "x") + "w0d_8_26_5" * COS(5 * 0.4 * "x");
    "phi" := "phi" + "w0c_8_26_6" * SIN(6 * 0.4 * "x") + "w0d_8_26_6" * COS(6 * 0.4 * "x");
    "acc" := "acc" + "phi";
    "x" := "feat_27";
    "phi" := "w0b_8_27" * "x" / (1.0 + EXP(-"x"));
    "phi" := "phi" + "w0c_8_27_1" * SIN(1 * 0.4 * "x") + "w0d_8_27_1" * COS(1 * 0.4 * "x");
    "phi" := "phi" + "w0c_8_27_2" * SIN(2 * 0.4 * "x") + "w0d_8_27_2" * COS(2 * 0.4 * "x");
    "phi" := "phi" + "w0c_8_27_3" * SIN(3 * 0.4 * "x") + "w0d_8_27_3" * COS(3 * 0.4 * "x");
    "phi" := "phi" + "w0c_8_27_4" * SIN(4 * 0.4 * "x") + "w0d_8_27_4" * COS(4 * 0.4 * "x");
    "phi" := "phi" + "w0c_8_27_5" * SIN(5 * 0.4 * "x") + "w0d_8_27_5" * COS(5 * 0.4 * "x");
    "phi" := "phi" + "w0c_8_27_6" * SIN(6 * 0.4 * "x") + "w0d_8_27_6" * COS(6 * 0.4 * "x");
    "acc" := "acc" + "phi";
    "x" := "feat_28";
    "phi" := "w0b_8_28" * "x" / (1.0 + EXP(-"x"));
    "phi" := "phi" + "w0c_8_28_1" * SIN(1 * 0.4 * "x") + "w0d_8_28_1" * COS(1 * 0.4 * "x");
    "phi" := "phi" + "w0c_8_28_2" * SIN(2 * 0.4 * "x") + "w0d_8_28_2" * COS(2 * 0.4 * "x");
    "phi" := "phi" + "w0c_8_28_3" * SIN(3 * 0.4 * "x") + "w0d_8_28_3" * COS(3 * 0.4 * "x");
    "phi" := "phi" + "w0c_8_28_4" * SIN(4 * 0.4 * "x") + "w0d_8_28_4" * COS(4 * 0.4 * "x");
    "phi" := "phi" + "w0c_8_28_5" * SIN(5 * 0.4 * "x") + "w0d_8_28_5" * COS(5 * 0.4 * "x");
    "phi" := "phi" + "w0c_8_28_6" * SIN(6 * 0.4 * "x") + "w0d_8_28_6" * COS(6 * 0.4 * "x");
    "acc" := "acc" + "phi";
    "h1_8" := "acc" + "b0_8";
    "acc" := 0.0;
    "x" := "feat_1";
    "phi" := "w0b_9_1" * "x" / (1.0 + EXP(-"x"));
    "phi" := "phi" + "w0c_9_1_1" * SIN(1 * 0.4 * "x") + "w0d_9_1_1" * COS(1 * 0.4 * "x");
    "phi" := "phi" + "w0c_9_1_2" * SIN(2 * 0.4 * "x") + "w0d_9_1_2" * COS(2 * 0.4 * "x");
    "phi" := "phi" + "w0c_9_1_3" * SIN(3 * 0.4 * "x") + "w0d_9_1_3" * COS(3 * 0.4 * "x");
    "phi" := "phi" + "w0c_9_1_4" * SIN(4 * 0.4 * "x") + "w0d_9_1_4" * COS(4 * 0.4 * "x");
    "phi" := "phi" + "w0c_9_1_5" * SIN(5 * 0.4 * "x") + "w0d_9_1_5" * COS(5 * 0.4 * "x");
    "phi" := "phi" + "w0c_9_1_6" * SIN(6 * 0.4 * "x") + "w0d_9_1_6" * COS(6 * 0.4 * "x");
    "acc" := "acc" + "phi";
    "x" := "feat_2";
    "phi" := "w0b_9_2" * "x" / (1.0 + EXP(-"x"));
    "phi" := "phi" + "w0c_9_2_1" * SIN(1 * 0.4 * "x") + "w0d_9_2_1" * COS(1 * 0.4 * "x");
    "phi" := "phi" + "w0c_9_2_2" * SIN(2 * 0.4 * "x") + "w0d_9_2_2" * COS(2 * 0.4 * "x");
    "phi" := "phi" + "w0c_9_2_3" * SIN(3 * 0.4 * "x") + "w0d_9_2_3" * COS(3 * 0.4 * "x");
    "phi" := "phi" + "w0c_9_2_4" * SIN(4 * 0.4 * "x") + "w0d_9_2_4" * COS(4 * 0.4 * "x");
    "phi" := "phi" + "w0c_9_2_5" * SIN(5 * 0.4 * "x") + "w0d_9_2_5" * COS(5 * 0.4 * "x");
    "phi" := "phi" + "w0c_9_2_6" * SIN(6 * 0.4 * "x") + "w0d_9_2_6" * COS(6 * 0.4 * "x");
    "acc" := "acc" + "phi";
    "x" := "feat_3";
    "phi" := "w0b_9_3" * "x" / (1.0 + EXP(-"x"));
    "phi" := "phi" + "w0c_9_3_1" * SIN(1 * 0.4 * "x") + "w0d_9_3_1" * COS(1 * 0.4 * "x");
    "phi" := "phi" + "w0c_9_3_2" * SIN(2 * 0.4 * "x") + "w0d_9_3_2" * COS(2 * 0.4 * "x");
    "phi" := "phi" + "w0c_9_3_3" * SIN(3 * 0.4 * "x") + "w0d_9_3_3" * COS(3 * 0.4 * "x");
    "phi" := "phi" + "w0c_9_3_4" * SIN(4 * 0.4 * "x") + "w0d_9_3_4" * COS(4 * 0.4 * "x");
    "phi" := "phi" + "w0c_9_3_5" * SIN(5 * 0.4 * "x") + "w0d_9_3_5" * COS(5 * 0.4 * "x");
    "phi" := "phi" + "w0c_9_3_6" * SIN(6 * 0.4 * "x") + "w0d_9_3_6" * COS(6 * 0.4 * "x");
    "acc" := "acc" + "phi";
    "x" := "feat_4";
    "phi" := "w0b_9_4" * "x" / (1.0 + EXP(-"x"));
    "phi" := "phi" + "w0c_9_4_1" * SIN(1 * 0.4 * "x") + "w0d_9_4_1" * COS(1 * 0.4 * "x");
    "phi" := "phi" + "w0c_9_4_2" * SIN(2 * 0.4 * "x") + "w0d_9_4_2" * COS(2 * 0.4 * "x");
    "phi" := "phi" + "w0c_9_4_3" * SIN(3 * 0.4 * "x") + "w0d_9_4_3" * COS(3 * 0.4 * "x");
    "phi" := "phi" + "w0c_9_4_4" * SIN(4 * 0.4 * "x") + "w0d_9_4_4" * COS(4 * 0.4 * "x");
    "phi" := "phi" + "w0c_9_4_5" * SIN(5 * 0.4 * "x") + "w0d_9_4_5" * COS(5 * 0.4 * "x");
    "phi" := "phi" + "w0c_9_4_6" * SIN(6 * 0.4 * "x") + "w0d_9_4_6" * COS(6 * 0.4 * "x");
    "acc" := "acc" + "phi";
    "x" := "feat_5";
    "phi" := "w0b_9_5" * "x" / (1.0 + EXP(-"x"));
    "phi" := "phi" + "w0c_9_5_1" * SIN(1 * 0.4 * "x") + "w0d_9_5_1" * COS(1 * 0.4 * "x");
    "phi" := "phi" + "w0c_9_5_2" * SIN(2 * 0.4 * "x") + "w0d_9_5_2" * COS(2 * 0.4 * "x");
    "phi" := "phi" + "w0c_9_5_3" * SIN(3 * 0.4 * "x") + "w0d_9_5_3" * COS(3 * 0.4 * "x");
    "phi" := "phi" + "w0c_9_5_4" * SIN(4 * 0.4 * "x") + "w0d_9_5_4" * COS(4 * 0.4 * "x");
    "phi" := "phi" + "w0c_9_5_5" * SIN(5 * 0.4 * "x") + "w0d_9_5_5" * COS(5 * 0.4 * "x");
    "phi" := "phi" + "w0c_9_5_6" * SIN(6 * 0.4 * "x") + "w0d_9_5_6" * COS(6 * 0.4 * "x");
    "acc" := "acc" + "phi";
    "x" := "feat_6";
    "phi" := "w0b_9_6" * "x" / (1.0 + EXP(-"x"));
    "phi" := "phi" + "w0c_9_6_1" * SIN(1 * 0.4 * "x") + "w0d_9_6_1" * COS(1 * 0.4 * "x");
    "phi" := "phi" + "w0c_9_6_2" * SIN(2 * 0.4 * "x") + "w0d_9_6_2" * COS(2 * 0.4 * "x");
    "phi" := "phi" + "w0c_9_6_3" * SIN(3 * 0.4 * "x") + "w0d_9_6_3" * COS(3 * 0.4 * "x");
    "phi" := "phi" + "w0c_9_6_4" * SIN(4 * 0.4 * "x") + "w0d_9_6_4" * COS(4 * 0.4 * "x");
    "phi" := "phi" + "w0c_9_6_5" * SIN(5 * 0.4 * "x") + "w0d_9_6_5" * COS(5 * 0.4 * "x");
    "phi" := "phi" + "w0c_9_6_6" * SIN(6 * 0.4 * "x") + "w0d_9_6_6" * COS(6 * 0.4 * "x");
    "acc" := "acc" + "phi";
    "x" := "feat_7";
    "phi" := "w0b_9_7" * "x" / (1.0 + EXP(-"x"));
    "phi" := "phi" + "w0c_9_7_1" * SIN(1 * 0.4 * "x") + "w0d_9_7_1" * COS(1 * 0.4 * "x");
    "phi" := "phi" + "w0c_9_7_2" * SIN(2 * 0.4 * "x") + "w0d_9_7_2" * COS(2 * 0.4 * "x");
    "phi" := "phi" + "w0c_9_7_3" * SIN(3 * 0.4 * "x") + "w0d_9_7_3" * COS(3 * 0.4 * "x");
    "phi" := "phi" + "w0c_9_7_4" * SIN(4 * 0.4 * "x") + "w0d_9_7_4" * COS(4 * 0.4 * "x");
    "phi" := "phi" + "w0c_9_7_5" * SIN(5 * 0.4 * "x") + "w0d_9_7_5" * COS(5 * 0.4 * "x");
    "phi" := "phi" + "w0c_9_7_6" * SIN(6 * 0.4 * "x") + "w0d_9_7_6" * COS(6 * 0.4 * "x");
    "acc" := "acc" + "phi";
    "x" := "feat_8";
    "phi" := "w0b_9_8" * "x" / (1.0 + EXP(-"x"));
    "phi" := "phi" + "w0c_9_8_1" * SIN(1 * 0.4 * "x") + "w0d_9_8_1" * COS(1 * 0.4 * "x");
    "phi" := "phi" + "w0c_9_8_2" * SIN(2 * 0.4 * "x") + "w0d_9_8_2" * COS(2 * 0.4 * "x");
    "phi" := "phi" + "w0c_9_8_3" * SIN(3 * 0.4 * "x") + "w0d_9_8_3" * COS(3 * 0.4 * "x");
    "phi" := "phi" + "w0c_9_8_4" * SIN(4 * 0.4 * "x") + "w0d_9_8_4" * COS(4 * 0.4 * "x");
    "phi" := "phi" + "w0c_9_8_5" * SIN(5 * 0.4 * "x") + "w0d_9_8_5" * COS(5 * 0.4 * "x");
    "phi" := "phi" + "w0c_9_8_6" * SIN(6 * 0.4 * "x") + "w0d_9_8_6" * COS(6 * 0.4 * "x");
    "acc" := "acc" + "phi";
    "x" := "feat_9";
    "phi" := "w0b_9_9" * "x" / (1.0 + EXP(-"x"));
    "phi" := "phi" + "w0c_9_9_1" * SIN(1 * 0.4 * "x") + "w0d_9_9_1" * COS(1 * 0.4 * "x");
    "phi" := "phi" + "w0c_9_9_2" * SIN(2 * 0.4 * "x") + "w0d_9_9_2" * COS(2 * 0.4 * "x");
    "phi" := "phi" + "w0c_9_9_3" * SIN(3 * 0.4 * "x") + "w0d_9_9_3" * COS(3 * 0.4 * "x");
    "phi" := "phi" + "w0c_9_9_4" * SIN(4 * 0.4 * "x") + "w0d_9_9_4" * COS(4 * 0.4 * "x");
    "phi" := "phi" + "w0c_9_9_5" * SIN(5 * 0.4 * "x") + "w0d_9_9_5" * COS(5 * 0.4 * "x");
    "phi" := "phi" + "w0c_9_9_6" * SIN(6 * 0.4 * "x") + "w0d_9_9_6" * COS(6 * 0.4 * "x");
    "acc" := "acc" + "phi";
    "x" := "feat_10";
    "phi" := "w0b_9_10" * "x" / (1.0 + EXP(-"x"));
    "phi" := "phi" + "w0c_9_10_1" * SIN(1 * 0.4 * "x") + "w0d_9_10_1" * COS(1 * 0.4 * "x");
    "phi" := "phi" + "w0c_9_10_2" * SIN(2 * 0.4 * "x") + "w0d_9_10_2" * COS(2 * 0.4 * "x");
    "phi" := "phi" + "w0c_9_10_3" * SIN(3 * 0.4 * "x") + "w0d_9_10_3" * COS(3 * 0.4 * "x");
    "phi" := "phi" + "w0c_9_10_4" * SIN(4 * 0.4 * "x") + "w0d_9_10_4" * COS(4 * 0.4 * "x");
    "phi" := "phi" + "w0c_9_10_5" * SIN(5 * 0.4 * "x") + "w0d_9_10_5" * COS(5 * 0.4 * "x");
    "phi" := "phi" + "w0c_9_10_6" * SIN(6 * 0.4 * "x") + "w0d_9_10_6" * COS(6 * 0.4 * "x");
    "acc" := "acc" + "phi";
    "x" := "feat_11";
    "phi" := "w0b_9_11" * "x" / (1.0 + EXP(-"x"));
    "phi" := "phi" + "w0c_9_11_1" * SIN(1 * 0.4 * "x") + "w0d_9_11_1" * COS(1 * 0.4 * "x");
    "phi" := "phi" + "w0c_9_11_2" * SIN(2 * 0.4 * "x") + "w0d_9_11_2" * COS(2 * 0.4 * "x");
    "phi" := "phi" + "w0c_9_11_3" * SIN(3 * 0.4 * "x") + "w0d_9_11_3" * COS(3 * 0.4 * "x");
    "phi" := "phi" + "w0c_9_11_4" * SIN(4 * 0.4 * "x") + "w0d_9_11_4" * COS(4 * 0.4 * "x");
    "phi" := "phi" + "w0c_9_11_5" * SIN(5 * 0.4 * "x") + "w0d_9_11_5" * COS(5 * 0.4 * "x");
    "phi" := "phi" + "w0c_9_11_6" * SIN(6 * 0.4 * "x") + "w0d_9_11_6" * COS(6 * 0.4 * "x");
    "acc" := "acc" + "phi";
    "x" := "feat_12";
    "phi" := "w0b_9_12" * "x" / (1.0 + EXP(-"x"));
    "phi" := "phi" + "w0c_9_12_1" * SIN(1 * 0.4 * "x") + "w0d_9_12_1" * COS(1 * 0.4 * "x");
    "phi" := "phi" + "w0c_9_12_2" * SIN(2 * 0.4 * "x") + "w0d_9_12_2" * COS(2 * 0.4 * "x");
    "phi" := "phi" + "w0c_9_12_3" * SIN(3 * 0.4 * "x") + "w0d_9_12_3" * COS(3 * 0.4 * "x");
    "phi" := "phi" + "w0c_9_12_4" * SIN(4 * 0.4 * "x") + "w0d_9_12_4" * COS(4 * 0.4 * "x");
    "phi" := "phi" + "w0c_9_12_5" * SIN(5 * 0.4 * "x") + "w0d_9_12_5" * COS(5 * 0.4 * "x");
    "phi" := "phi" + "w0c_9_12_6" * SIN(6 * 0.4 * "x") + "w0d_9_12_6" * COS(6 * 0.4 * "x");
    "acc" := "acc" + "phi";
    "x" := "feat_13";
    "phi" := "w0b_9_13" * "x" / (1.0 + EXP(-"x"));
    "phi" := "phi" + "w0c_9_13_1" * SIN(1 * 0.4 * "x") + "w0d_9_13_1" * COS(1 * 0.4 * "x");
    "phi" := "phi" + "w0c_9_13_2" * SIN(2 * 0.4 * "x") + "w0d_9_13_2" * COS(2 * 0.4 * "x");
    "phi" := "phi" + "w0c_9_13_3" * SIN(3 * 0.4 * "x") + "w0d_9_13_3" * COS(3 * 0.4 * "x");
    "phi" := "phi" + "w0c_9_13_4" * SIN(4 * 0.4 * "x") + "w0d_9_13_4" * COS(4 * 0.4 * "x");
    "phi" := "phi" + "w0c_9_13_5" * SIN(5 * 0.4 * "x") + "w0d_9_13_5" * COS(5 * 0.4 * "x");
    "phi" := "phi" + "w0c_9_13_6" * SIN(6 * 0.4 * "x") + "w0d_9_13_6" * COS(6 * 0.4 * "x");
    "acc" := "acc" + "phi";
    "x" := "feat_14";
    "phi" := "w0b_9_14" * "x" / (1.0 + EXP(-"x"));
    "phi" := "phi" + "w0c_9_14_1" * SIN(1 * 0.4 * "x") + "w0d_9_14_1" * COS(1 * 0.4 * "x");
    "phi" := "phi" + "w0c_9_14_2" * SIN(2 * 0.4 * "x") + "w0d_9_14_2" * COS(2 * 0.4 * "x");
    "phi" := "phi" + "w0c_9_14_3" * SIN(3 * 0.4 * "x") + "w0d_9_14_3" * COS(3 * 0.4 * "x");
    "phi" := "phi" + "w0c_9_14_4" * SIN(4 * 0.4 * "x") + "w0d_9_14_4" * COS(4 * 0.4 * "x");
    "phi" := "phi" + "w0c_9_14_5" * SIN(5 * 0.4 * "x") + "w0d_9_14_5" * COS(5 * 0.4 * "x");
    "phi" := "phi" + "w0c_9_14_6" * SIN(6 * 0.4 * "x") + "w0d_9_14_6" * COS(6 * 0.4 * "x");
    "acc" := "acc" + "phi";
    "x" := "feat_15";
    "phi" := "w0b_9_15" * "x" / (1.0 + EXP(-"x"));
    "phi" := "phi" + "w0c_9_15_1" * SIN(1 * 0.4 * "x") + "w0d_9_15_1" * COS(1 * 0.4 * "x");
    "phi" := "phi" + "w0c_9_15_2" * SIN(2 * 0.4 * "x") + "w0d_9_15_2" * COS(2 * 0.4 * "x");
    "phi" := "phi" + "w0c_9_15_3" * SIN(3 * 0.4 * "x") + "w0d_9_15_3" * COS(3 * 0.4 * "x");
    "phi" := "phi" + "w0c_9_15_4" * SIN(4 * 0.4 * "x") + "w0d_9_15_4" * COS(4 * 0.4 * "x");
    "phi" := "phi" + "w0c_9_15_5" * SIN(5 * 0.4 * "x") + "w0d_9_15_5" * COS(5 * 0.4 * "x");
    "phi" := "phi" + "w0c_9_15_6" * SIN(6 * 0.4 * "x") + "w0d_9_15_6" * COS(6 * 0.4 * "x");
    "acc" := "acc" + "phi";
    "x" := "feat_16";
    "phi" := "w0b_9_16" * "x" / (1.0 + EXP(-"x"));
    "phi" := "phi" + "w0c_9_16_1" * SIN(1 * 0.4 * "x") + "w0d_9_16_1" * COS(1 * 0.4 * "x");
    "phi" := "phi" + "w0c_9_16_2" * SIN(2 * 0.4 * "x") + "w0d_9_16_2" * COS(2 * 0.4 * "x");
    "phi" := "phi" + "w0c_9_16_3" * SIN(3 * 0.4 * "x") + "w0d_9_16_3" * COS(3 * 0.4 * "x");
    "phi" := "phi" + "w0c_9_16_4" * SIN(4 * 0.4 * "x") + "w0d_9_16_4" * COS(4 * 0.4 * "x");
    "phi" := "phi" + "w0c_9_16_5" * SIN(5 * 0.4 * "x") + "w0d_9_16_5" * COS(5 * 0.4 * "x");
    "phi" := "phi" + "w0c_9_16_6" * SIN(6 * 0.4 * "x") + "w0d_9_16_6" * COS(6 * 0.4 * "x");
    "acc" := "acc" + "phi";
    "x" := "feat_17";
    "phi" := "w0b_9_17" * "x" / (1.0 + EXP(-"x"));
    "phi" := "phi" + "w0c_9_17_1" * SIN(1 * 0.4 * "x") + "w0d_9_17_1" * COS(1 * 0.4 * "x");
    "phi" := "phi" + "w0c_9_17_2" * SIN(2 * 0.4 * "x") + "w0d_9_17_2" * COS(2 * 0.4 * "x");
    "phi" := "phi" + "w0c_9_17_3" * SIN(3 * 0.4 * "x") + "w0d_9_17_3" * COS(3 * 0.4 * "x");
    "phi" := "phi" + "w0c_9_17_4" * SIN(4 * 0.4 * "x") + "w0d_9_17_4" * COS(4 * 0.4 * "x");
    "phi" := "phi" + "w0c_9_17_5" * SIN(5 * 0.4 * "x") + "w0d_9_17_5" * COS(5 * 0.4 * "x");
    "phi" := "phi" + "w0c_9_17_6" * SIN(6 * 0.4 * "x") + "w0d_9_17_6" * COS(6 * 0.4 * "x");
    "acc" := "acc" + "phi";
    "x" := "feat_18";
    "phi" := "w0b_9_18" * "x" / (1.0 + EXP(-"x"));
    "phi" := "phi" + "w0c_9_18_1" * SIN(1 * 0.4 * "x") + "w0d_9_18_1" * COS(1 * 0.4 * "x");
    "phi" := "phi" + "w0c_9_18_2" * SIN(2 * 0.4 * "x") + "w0d_9_18_2" * COS(2 * 0.4 * "x");
    "phi" := "phi" + "w0c_9_18_3" * SIN(3 * 0.4 * "x") + "w0d_9_18_3" * COS(3 * 0.4 * "x");
    "phi" := "phi" + "w0c_9_18_4" * SIN(4 * 0.4 * "x") + "w0d_9_18_4" * COS(4 * 0.4 * "x");
    "phi" := "phi" + "w0c_9_18_5" * SIN(5 * 0.4 * "x") + "w0d_9_18_5" * COS(5 * 0.4 * "x");
    "phi" := "phi" + "w0c_9_18_6" * SIN(6 * 0.4 * "x") + "w0d_9_18_6" * COS(6 * 0.4 * "x");
    "acc" := "acc" + "phi";
    "x" := "feat_19";
    "phi" := "w0b_9_19" * "x" / (1.0 + EXP(-"x"));
    "phi" := "phi" + "w0c_9_19_1" * SIN(1 * 0.4 * "x") + "w0d_9_19_1" * COS(1 * 0.4 * "x");
    "phi" := "phi" + "w0c_9_19_2" * SIN(2 * 0.4 * "x") + "w0d_9_19_2" * COS(2 * 0.4 * "x");
    "phi" := "phi" + "w0c_9_19_3" * SIN(3 * 0.4 * "x") + "w0d_9_19_3" * COS(3 * 0.4 * "x");
    "phi" := "phi" + "w0c_9_19_4" * SIN(4 * 0.4 * "x") + "w0d_9_19_4" * COS(4 * 0.4 * "x");
    "phi" := "phi" + "w0c_9_19_5" * SIN(5 * 0.4 * "x") + "w0d_9_19_5" * COS(5 * 0.4 * "x");
    "phi" := "phi" + "w0c_9_19_6" * SIN(6 * 0.4 * "x") + "w0d_9_19_6" * COS(6 * 0.4 * "x");
    "acc" := "acc" + "phi";
    "x" := "feat_20";
    "phi" := "w0b_9_20" * "x" / (1.0 + EXP(-"x"));
    "phi" := "phi" + "w0c_9_20_1" * SIN(1 * 0.4 * "x") + "w0d_9_20_1" * COS(1 * 0.4 * "x");
    "phi" := "phi" + "w0c_9_20_2" * SIN(2 * 0.4 * "x") + "w0d_9_20_2" * COS(2 * 0.4 * "x");
    "phi" := "phi" + "w0c_9_20_3" * SIN(3 * 0.4 * "x") + "w0d_9_20_3" * COS(3 * 0.4 * "x");
    "phi" := "phi" + "w0c_9_20_4" * SIN(4 * 0.4 * "x") + "w0d_9_20_4" * COS(4 * 0.4 * "x");
    "phi" := "phi" + "w0c_9_20_5" * SIN(5 * 0.4 * "x") + "w0d_9_20_5" * COS(5 * 0.4 * "x");
    "phi" := "phi" + "w0c_9_20_6" * SIN(6 * 0.4 * "x") + "w0d_9_20_6" * COS(6 * 0.4 * "x");
    "acc" := "acc" + "phi";
    "x" := "feat_21";
    "phi" := "w0b_9_21" * "x" / (1.0 + EXP(-"x"));
    "phi" := "phi" + "w0c_9_21_1" * SIN(1 * 0.4 * "x") + "w0d_9_21_1" * COS(1 * 0.4 * "x");
    "phi" := "phi" + "w0c_9_21_2" * SIN(2 * 0.4 * "x") + "w0d_9_21_2" * COS(2 * 0.4 * "x");
    "phi" := "phi" + "w0c_9_21_3" * SIN(3 * 0.4 * "x") + "w0d_9_21_3" * COS(3 * 0.4 * "x");
    "phi" := "phi" + "w0c_9_21_4" * SIN(4 * 0.4 * "x") + "w0d_9_21_4" * COS(4 * 0.4 * "x");
    "phi" := "phi" + "w0c_9_21_5" * SIN(5 * 0.4 * "x") + "w0d_9_21_5" * COS(5 * 0.4 * "x");
    "phi" := "phi" + "w0c_9_21_6" * SIN(6 * 0.4 * "x") + "w0d_9_21_6" * COS(6 * 0.4 * "x");
    "acc" := "acc" + "phi";
    "x" := "feat_22";
    "phi" := "w0b_9_22" * "x" / (1.0 + EXP(-"x"));
    "phi" := "phi" + "w0c_9_22_1" * SIN(1 * 0.4 * "x") + "w0d_9_22_1" * COS(1 * 0.4 * "x");
    "phi" := "phi" + "w0c_9_22_2" * SIN(2 * 0.4 * "x") + "w0d_9_22_2" * COS(2 * 0.4 * "x");
    "phi" := "phi" + "w0c_9_22_3" * SIN(3 * 0.4 * "x") + "w0d_9_22_3" * COS(3 * 0.4 * "x");
    "phi" := "phi" + "w0c_9_22_4" * SIN(4 * 0.4 * "x") + "w0d_9_22_4" * COS(4 * 0.4 * "x");
    "phi" := "phi" + "w0c_9_22_5" * SIN(5 * 0.4 * "x") + "w0d_9_22_5" * COS(5 * 0.4 * "x");
    "phi" := "phi" + "w0c_9_22_6" * SIN(6 * 0.4 * "x") + "w0d_9_22_6" * COS(6 * 0.4 * "x");
    "acc" := "acc" + "phi";
    "x" := "feat_23";
    "phi" := "w0b_9_23" * "x" / (1.0 + EXP(-"x"));
    "phi" := "phi" + "w0c_9_23_1" * SIN(1 * 0.4 * "x") + "w0d_9_23_1" * COS(1 * 0.4 * "x");
    "phi" := "phi" + "w0c_9_23_2" * SIN(2 * 0.4 * "x") + "w0d_9_23_2" * COS(2 * 0.4 * "x");
    "phi" := "phi" + "w0c_9_23_3" * SIN(3 * 0.4 * "x") + "w0d_9_23_3" * COS(3 * 0.4 * "x");
    "phi" := "phi" + "w0c_9_23_4" * SIN(4 * 0.4 * "x") + "w0d_9_23_4" * COS(4 * 0.4 * "x");
    "phi" := "phi" + "w0c_9_23_5" * SIN(5 * 0.4 * "x") + "w0d_9_23_5" * COS(5 * 0.4 * "x");
    "phi" := "phi" + "w0c_9_23_6" * SIN(6 * 0.4 * "x") + "w0d_9_23_6" * COS(6 * 0.4 * "x");
    "acc" := "acc" + "phi";
    "x" := "feat_24";
    "phi" := "w0b_9_24" * "x" / (1.0 + EXP(-"x"));
    "phi" := "phi" + "w0c_9_24_1" * SIN(1 * 0.4 * "x") + "w0d_9_24_1" * COS(1 * 0.4 * "x");
    "phi" := "phi" + "w0c_9_24_2" * SIN(2 * 0.4 * "x") + "w0d_9_24_2" * COS(2 * 0.4 * "x");
    "phi" := "phi" + "w0c_9_24_3" * SIN(3 * 0.4 * "x") + "w0d_9_24_3" * COS(3 * 0.4 * "x");
    "phi" := "phi" + "w0c_9_24_4" * SIN(4 * 0.4 * "x") + "w0d_9_24_4" * COS(4 * 0.4 * "x");
    "phi" := "phi" + "w0c_9_24_5" * SIN(5 * 0.4 * "x") + "w0d_9_24_5" * COS(5 * 0.4 * "x");
    "phi" := "phi" + "w0c_9_24_6" * SIN(6 * 0.4 * "x") + "w0d_9_24_6" * COS(6 * 0.4 * "x");
    "acc" := "acc" + "phi";
    "x" := "feat_25";
    "phi" := "w0b_9_25" * "x" / (1.0 + EXP(-"x"));
    "phi" := "phi" + "w0c_9_25_1" * SIN(1 * 0.4 * "x") + "w0d_9_25_1" * COS(1 * 0.4 * "x");
    "phi" := "phi" + "w0c_9_25_2" * SIN(2 * 0.4 * "x") + "w0d_9_25_2" * COS(2 * 0.4 * "x");
    "phi" := "phi" + "w0c_9_25_3" * SIN(3 * 0.4 * "x") + "w0d_9_25_3" * COS(3 * 0.4 * "x");
    "phi" := "phi" + "w0c_9_25_4" * SIN(4 * 0.4 * "x") + "w0d_9_25_4" * COS(4 * 0.4 * "x");
    "phi" := "phi" + "w0c_9_25_5" * SIN(5 * 0.4 * "x") + "w0d_9_25_5" * COS(5 * 0.4 * "x");
    "phi" := "phi" + "w0c_9_25_6" * SIN(6 * 0.4 * "x") + "w0d_9_25_6" * COS(6 * 0.4 * "x");
    "acc" := "acc" + "phi";
    "x" := "feat_26";
    "phi" := "w0b_9_26" * "x" / (1.0 + EXP(-"x"));
    "phi" := "phi" + "w0c_9_26_1" * SIN(1 * 0.4 * "x") + "w0d_9_26_1" * COS(1 * 0.4 * "x");
    "phi" := "phi" + "w0c_9_26_2" * SIN(2 * 0.4 * "x") + "w0d_9_26_2" * COS(2 * 0.4 * "x");
    "phi" := "phi" + "w0c_9_26_3" * SIN(3 * 0.4 * "x") + "w0d_9_26_3" * COS(3 * 0.4 * "x");
    "phi" := "phi" + "w0c_9_26_4" * SIN(4 * 0.4 * "x") + "w0d_9_26_4" * COS(4 * 0.4 * "x");
    "phi" := "phi" + "w0c_9_26_5" * SIN(5 * 0.4 * "x") + "w0d_9_26_5" * COS(5 * 0.4 * "x");
    "phi" := "phi" + "w0c_9_26_6" * SIN(6 * 0.4 * "x") + "w0d_9_26_6" * COS(6 * 0.4 * "x");
    "acc" := "acc" + "phi";
    "x" := "feat_27";
    "phi" := "w0b_9_27" * "x" / (1.0 + EXP(-"x"));
    "phi" := "phi" + "w0c_9_27_1" * SIN(1 * 0.4 * "x") + "w0d_9_27_1" * COS(1 * 0.4 * "x");
    "phi" := "phi" + "w0c_9_27_2" * SIN(2 * 0.4 * "x") + "w0d_9_27_2" * COS(2 * 0.4 * "x");
    "phi" := "phi" + "w0c_9_27_3" * SIN(3 * 0.4 * "x") + "w0d_9_27_3" * COS(3 * 0.4 * "x");
    "phi" := "phi" + "w0c_9_27_4" * SIN(4 * 0.4 * "x") + "w0d_9_27_4" * COS(4 * 0.4 * "x");
    "phi" := "phi" + "w0c_9_27_5" * SIN(5 * 0.4 * "x") + "w0d_9_27_5" * COS(5 * 0.4 * "x");
    "phi" := "phi" + "w0c_9_27_6" * SIN(6 * 0.4 * "x") + "w0d_9_27_6" * COS(6 * 0.4 * "x");
    "acc" := "acc" + "phi";
    "x" := "feat_28";
    "phi" := "w0b_9_28" * "x" / (1.0 + EXP(-"x"));
    "phi" := "phi" + "w0c_9_28_1" * SIN(1 * 0.4 * "x") + "w0d_9_28_1" * COS(1 * 0.4 * "x");
    "phi" := "phi" + "w0c_9_28_2" * SIN(2 * 0.4 * "x") + "w0d_9_28_2" * COS(2 * 0.4 * "x");
    "phi" := "phi" + "w0c_9_28_3" * SIN(3 * 0.4 * "x") + "w0d_9_28_3" * COS(3 * 0.4 * "x");
    "phi" := "phi" + "w0c_9_28_4" * SIN(4 * 0.4 * "x") + "w0d_9_28_4" * COS(4 * 0.4 * "x");
    "phi" := "phi" + "w0c_9_28_5" * SIN(5 * 0.4 * "x") + "w0d_9_28_5" * COS(5 * 0.4 * "x");
    "phi" := "phi" + "w0c_9_28_6" * SIN(6 * 0.4 * "x") + "w0d_9_28_6" * COS(6 * 0.4 * "x");
    "acc" := "acc" + "phi";
    "h1_9" := "acc" + "b0_9";
    "acc" := 0.0;
    "x" := "feat_1";
    "phi" := "w0b_10_1" * "x" / (1.0 + EXP(-"x"));
    "phi" := "phi" + "w0c_10_1_1" * SIN(1 * 0.4 * "x") + "w0d_10_1_1" * COS(1 * 0.4 * "x");
    "phi" := "phi" + "w0c_10_1_2" * SIN(2 * 0.4 * "x") + "w0d_10_1_2" * COS(2 * 0.4 * "x");
    "phi" := "phi" + "w0c_10_1_3" * SIN(3 * 0.4 * "x") + "w0d_10_1_3" * COS(3 * 0.4 * "x");
    "phi" := "phi" + "w0c_10_1_4" * SIN(4 * 0.4 * "x") + "w0d_10_1_4" * COS(4 * 0.4 * "x");
    "phi" := "phi" + "w0c_10_1_5" * SIN(5 * 0.4 * "x") + "w0d_10_1_5" * COS(5 * 0.4 * "x");
    "phi" := "phi" + "w0c_10_1_6" * SIN(6 * 0.4 * "x") + "w0d_10_1_6" * COS(6 * 0.4 * "x");
    "acc" := "acc" + "phi";
    "x" := "feat_2";
    "phi" := "w0b_10_2" * "x" / (1.0 + EXP(-"x"));
    "phi" := "phi" + "w0c_10_2_1" * SIN(1 * 0.4 * "x") + "w0d_10_2_1" * COS(1 * 0.4 * "x");
    "phi" := "phi" + "w0c_10_2_2" * SIN(2 * 0.4 * "x") + "w0d_10_2_2" * COS(2 * 0.4 * "x");
    "phi" := "phi" + "w0c_10_2_3" * SIN(3 * 0.4 * "x") + "w0d_10_2_3" * COS(3 * 0.4 * "x");
    "phi" := "phi" + "w0c_10_2_4" * SIN(4 * 0.4 * "x") + "w0d_10_2_4" * COS(4 * 0.4 * "x");
    "phi" := "phi" + "w0c_10_2_5" * SIN(5 * 0.4 * "x") + "w0d_10_2_5" * COS(5 * 0.4 * "x");
    "phi" := "phi" + "w0c_10_2_6" * SIN(6 * 0.4 * "x") + "w0d_10_2_6" * COS(6 * 0.4 * "x");
    "acc" := "acc" + "phi";
    "x" := "feat_3";
    "phi" := "w0b_10_3" * "x" / (1.0 + EXP(-"x"));
    "phi" := "phi" + "w0c_10_3_1" * SIN(1 * 0.4 * "x") + "w0d_10_3_1" * COS(1 * 0.4 * "x");
    "phi" := "phi" + "w0c_10_3_2" * SIN(2 * 0.4 * "x") + "w0d_10_3_2" * COS(2 * 0.4 * "x");
    "phi" := "phi" + "w0c_10_3_3" * SIN(3 * 0.4 * "x") + "w0d_10_3_3" * COS(3 * 0.4 * "x");
    "phi" := "phi" + "w0c_10_3_4" * SIN(4 * 0.4 * "x") + "w0d_10_3_4" * COS(4 * 0.4 * "x");
    "phi" := "phi" + "w0c_10_3_5" * SIN(5 * 0.4 * "x") + "w0d_10_3_5" * COS(5 * 0.4 * "x");
    "phi" := "phi" + "w0c_10_3_6" * SIN(6 * 0.4 * "x") + "w0d_10_3_6" * COS(6 * 0.4 * "x");
    "acc" := "acc" + "phi";
    "x" := "feat_4";
    "phi" := "w0b_10_4" * "x" / (1.0 + EXP(-"x"));
    "phi" := "phi" + "w0c_10_4_1" * SIN(1 * 0.4 * "x") + "w0d_10_4_1" * COS(1 * 0.4 * "x");
    "phi" := "phi" + "w0c_10_4_2" * SIN(2 * 0.4 * "x") + "w0d_10_4_2" * COS(2 * 0.4 * "x");
    "phi" := "phi" + "w0c_10_4_3" * SIN(3 * 0.4 * "x") + "w0d_10_4_3" * COS(3 * 0.4 * "x");
    "phi" := "phi" + "w0c_10_4_4" * SIN(4 * 0.4 * "x") + "w0d_10_4_4" * COS(4 * 0.4 * "x");
    "phi" := "phi" + "w0c_10_4_5" * SIN(5 * 0.4 * "x") + "w0d_10_4_5" * COS(5 * 0.4 * "x");
    "phi" := "phi" + "w0c_10_4_6" * SIN(6 * 0.4 * "x") + "w0d_10_4_6" * COS(6 * 0.4 * "x");
    "acc" := "acc" + "phi";
    "x" := "feat_5";
    "phi" := "w0b_10_5" * "x" / (1.0 + EXP(-"x"));
    "phi" := "phi" + "w0c_10_5_1" * SIN(1 * 0.4 * "x") + "w0d_10_5_1" * COS(1 * 0.4 * "x");
    "phi" := "phi" + "w0c_10_5_2" * SIN(2 * 0.4 * "x") + "w0d_10_5_2" * COS(2 * 0.4 * "x");
    "phi" := "phi" + "w0c_10_5_3" * SIN(3 * 0.4 * "x") + "w0d_10_5_3" * COS(3 * 0.4 * "x");
    "phi" := "phi" + "w0c_10_5_4" * SIN(4 * 0.4 * "x") + "w0d_10_5_4" * COS(4 * 0.4 * "x");
    "phi" := "phi" + "w0c_10_5_5" * SIN(5 * 0.4 * "x") + "w0d_10_5_5" * COS(5 * 0.4 * "x");
    "phi" := "phi" + "w0c_10_5_6" * SIN(6 * 0.4 * "x") + "w0d_10_5_6" * COS(6 * 0.4 * "x");
    "acc" := "acc" + "phi";
    "x" := "feat_6";
    "phi" := "w0b_10_6" * "x" / (1.0 + EXP(-"x"));
    "phi" := "phi" + "w0c_10_6_1" * SIN(1 * 0.4 * "x") + "w0d_10_6_1" * COS(1 * 0.4 * "x");
    "phi" := "phi" + "w0c_10_6_2" * SIN(2 * 0.4 * "x") + "w0d_10_6_2" * COS(2 * 0.4 * "x");
    "phi" := "phi" + "w0c_10_6_3" * SIN(3 * 0.4 * "x") + "w0d_10_6_3" * COS(3 * 0.4 * "x");
    "phi" := "phi" + "w0c_10_6_4" * SIN(4 * 0.4 * "x") + "w0d_10_6_4" * COS(4 * 0.4 * "x");
    "phi" := "phi" + "w0c_10_6_5" * SIN(5 * 0.4 * "x") + "w0d_10_6_5" * COS(5 * 0.4 * "x");
    "phi" := "phi" + "w0c_10_6_6" * SIN(6 * 0.4 * "x") + "w0d_10_6_6" * COS(6 * 0.4 * "x");
    "acc" := "acc" + "phi";
    "x" := "feat_7";
    "phi" := "w0b_10_7" * "x" / (1.0 + EXP(-"x"));
    "phi" := "phi" + "w0c_10_7_1" * SIN(1 * 0.4 * "x") + "w0d_10_7_1" * COS(1 * 0.4 * "x");
    "phi" := "phi" + "w0c_10_7_2" * SIN(2 * 0.4 * "x") + "w0d_10_7_2" * COS(2 * 0.4 * "x");
    "phi" := "phi" + "w0c_10_7_3" * SIN(3 * 0.4 * "x") + "w0d_10_7_3" * COS(3 * 0.4 * "x");
    "phi" := "phi" + "w0c_10_7_4" * SIN(4 * 0.4 * "x") + "w0d_10_7_4" * COS(4 * 0.4 * "x");
    "phi" := "phi" + "w0c_10_7_5" * SIN(5 * 0.4 * "x") + "w0d_10_7_5" * COS(5 * 0.4 * "x");
    "phi" := "phi" + "w0c_10_7_6" * SIN(6 * 0.4 * "x") + "w0d_10_7_6" * COS(6 * 0.4 * "x");
    "acc" := "acc" + "phi";
    "x" := "feat_8";
    "phi" := "w0b_10_8" * "x" / (1.0 + EXP(-"x"));
    "phi" := "phi" + "w0c_10_8_1" * SIN(1 * 0.4 * "x") + "w0d_10_8_1" * COS(1 * 0.4 * "x");
    "phi" := "phi" + "w0c_10_8_2" * SIN(2 * 0.4 * "x") + "w0d_10_8_2" * COS(2 * 0.4 * "x");
    "phi" := "phi" + "w0c_10_8_3" * SIN(3 * 0.4 * "x") + "w0d_10_8_3" * COS(3 * 0.4 * "x");
    "phi" := "phi" + "w0c_10_8_4" * SIN(4 * 0.4 * "x") + "w0d_10_8_4" * COS(4 * 0.4 * "x");
    "phi" := "phi" + "w0c_10_8_5" * SIN(5 * 0.4 * "x") + "w0d_10_8_5" * COS(5 * 0.4 * "x");
    "phi" := "phi" + "w0c_10_8_6" * SIN(6 * 0.4 * "x") + "w0d_10_8_6" * COS(6 * 0.4 * "x");
    "acc" := "acc" + "phi";
    "x" := "feat_9";
    "phi" := "w0b_10_9" * "x" / (1.0 + EXP(-"x"));
    "phi" := "phi" + "w0c_10_9_1" * SIN(1 * 0.4 * "x") + "w0d_10_9_1" * COS(1 * 0.4 * "x");
    "phi" := "phi" + "w0c_10_9_2" * SIN(2 * 0.4 * "x") + "w0d_10_9_2" * COS(2 * 0.4 * "x");
    "phi" := "phi" + "w0c_10_9_3" * SIN(3 * 0.4 * "x") + "w0d_10_9_3" * COS(3 * 0.4 * "x");
    "phi" := "phi" + "w0c_10_9_4" * SIN(4 * 0.4 * "x") + "w0d_10_9_4" * COS(4 * 0.4 * "x");
    "phi" := "phi" + "w0c_10_9_5" * SIN(5 * 0.4 * "x") + "w0d_10_9_5" * COS(5 * 0.4 * "x");
    "phi" := "phi" + "w0c_10_9_6" * SIN(6 * 0.4 * "x") + "w0d_10_9_6" * COS(6 * 0.4 * "x");
    "acc" := "acc" + "phi";
    "x" := "feat_10";
    "phi" := "w0b_10_10" * "x" / (1.0 + EXP(-"x"));
    "phi" := "phi" + "w0c_10_10_1" * SIN(1 * 0.4 * "x") + "w0d_10_10_1" * COS(1 * 0.4 * "x");
    "phi" := "phi" + "w0c_10_10_2" * SIN(2 * 0.4 * "x") + "w0d_10_10_2" * COS(2 * 0.4 * "x");
    "phi" := "phi" + "w0c_10_10_3" * SIN(3 * 0.4 * "x") + "w0d_10_10_3" * COS(3 * 0.4 * "x");
    "phi" := "phi" + "w0c_10_10_4" * SIN(4 * 0.4 * "x") + "w0d_10_10_4" * COS(4 * 0.4 * "x");
    "phi" := "phi" + "w0c_10_10_5" * SIN(5 * 0.4 * "x") + "w0d_10_10_5" * COS(5 * 0.4 * "x");
    "phi" := "phi" + "w0c_10_10_6" * SIN(6 * 0.4 * "x") + "w0d_10_10_6" * COS(6 * 0.4 * "x");
    "acc" := "acc" + "phi";
    "x" := "feat_11";
    "phi" := "w0b_10_11" * "x" / (1.0 + EXP(-"x"));
    "phi" := "phi" + "w0c_10_11_1" * SIN(1 * 0.4 * "x") + "w0d_10_11_1" * COS(1 * 0.4 * "x");
    "phi" := "phi" + "w0c_10_11_2" * SIN(2 * 0.4 * "x") + "w0d_10_11_2" * COS(2 * 0.4 * "x");
    "phi" := "phi" + "w0c_10_11_3" * SIN(3 * 0.4 * "x") + "w0d_10_11_3" * COS(3 * 0.4 * "x");
    "phi" := "phi" + "w0c_10_11_4" * SIN(4 * 0.4 * "x") + "w0d_10_11_4" * COS(4 * 0.4 * "x");
    "phi" := "phi" + "w0c_10_11_5" * SIN(5 * 0.4 * "x") + "w0d_10_11_5" * COS(5 * 0.4 * "x");
    "phi" := "phi" + "w0c_10_11_6" * SIN(6 * 0.4 * "x") + "w0d_10_11_6" * COS(6 * 0.4 * "x");
    "acc" := "acc" + "phi";
    "x" := "feat_12";
    "phi" := "w0b_10_12" * "x" / (1.0 + EXP(-"x"));
    "phi" := "phi" + "w0c_10_12_1" * SIN(1 * 0.4 * "x") + "w0d_10_12_1" * COS(1 * 0.4 * "x");
    "phi" := "phi" + "w0c_10_12_2" * SIN(2 * 0.4 * "x") + "w0d_10_12_2" * COS(2 * 0.4 * "x");
    "phi" := "phi" + "w0c_10_12_3" * SIN(3 * 0.4 * "x") + "w0d_10_12_3" * COS(3 * 0.4 * "x");
    "phi" := "phi" + "w0c_10_12_4" * SIN(4 * 0.4 * "x") + "w0d_10_12_4" * COS(4 * 0.4 * "x");
    "phi" := "phi" + "w0c_10_12_5" * SIN(5 * 0.4 * "x") + "w0d_10_12_5" * COS(5 * 0.4 * "x");
    "phi" := "phi" + "w0c_10_12_6" * SIN(6 * 0.4 * "x") + "w0d_10_12_6" * COS(6 * 0.4 * "x");
    "acc" := "acc" + "phi";
    "x" := "feat_13";
    "phi" := "w0b_10_13" * "x" / (1.0 + EXP(-"x"));
    "phi" := "phi" + "w0c_10_13_1" * SIN(1 * 0.4 * "x") + "w0d_10_13_1" * COS(1 * 0.4 * "x");
    "phi" := "phi" + "w0c_10_13_2" * SIN(2 * 0.4 * "x") + "w0d_10_13_2" * COS(2 * 0.4 * "x");
    "phi" := "phi" + "w0c_10_13_3" * SIN(3 * 0.4 * "x") + "w0d_10_13_3" * COS(3 * 0.4 * "x");
    "phi" := "phi" + "w0c_10_13_4" * SIN(4 * 0.4 * "x") + "w0d_10_13_4" * COS(4 * 0.4 * "x");
    "phi" := "phi" + "w0c_10_13_5" * SIN(5 * 0.4 * "x") + "w0d_10_13_5" * COS(5 * 0.4 * "x");
    "phi" := "phi" + "w0c_10_13_6" * SIN(6 * 0.4 * "x") + "w0d_10_13_6" * COS(6 * 0.4 * "x");
    "acc" := "acc" + "phi";
    "x" := "feat_14";
    "phi" := "w0b_10_14" * "x" / (1.0 + EXP(-"x"));
    "phi" := "phi" + "w0c_10_14_1" * SIN(1 * 0.4 * "x") + "w0d_10_14_1" * COS(1 * 0.4 * "x");
    "phi" := "phi" + "w0c_10_14_2" * SIN(2 * 0.4 * "x") + "w0d_10_14_2" * COS(2 * 0.4 * "x");
    "phi" := "phi" + "w0c_10_14_3" * SIN(3 * 0.4 * "x") + "w0d_10_14_3" * COS(3 * 0.4 * "x");
    "phi" := "phi" + "w0c_10_14_4" * SIN(4 * 0.4 * "x") + "w0d_10_14_4" * COS(4 * 0.4 * "x");
    "phi" := "phi" + "w0c_10_14_5" * SIN(5 * 0.4 * "x") + "w0d_10_14_5" * COS(5 * 0.4 * "x");
    "phi" := "phi" + "w0c_10_14_6" * SIN(6 * 0.4 * "x") + "w0d_10_14_6" * COS(6 * 0.4 * "x");
    "acc" := "acc" + "phi";
    "x" := "feat_15";
    "phi" := "w0b_10_15" * "x" / (1.0 + EXP(-"x"));
    "phi" := "phi" + "w0c_10_15_1" * SIN(1 * 0.4 * "x") + "w0d_10_15_1" * COS(1 * 0.4 * "x");
    "phi" := "phi" + "w0c_10_15_2" * SIN(2 * 0.4 * "x") + "w0d_10_15_2" * COS(2 * 0.4 * "x");
    "phi" := "phi" + "w0c_10_15_3" * SIN(3 * 0.4 * "x") + "w0d_10_15_3" * COS(3 * 0.4 * "x");
    "phi" := "phi" + "w0c_10_15_4" * SIN(4 * 0.4 * "x") + "w0d_10_15_4" * COS(4 * 0.4 * "x");
    "phi" := "phi" + "w0c_10_15_5" * SIN(5 * 0.4 * "x") + "w0d_10_15_5" * COS(5 * 0.4 * "x");
    "phi" := "phi" + "w0c_10_15_6" * SIN(6 * 0.4 * "x") + "w0d_10_15_6" * COS(6 * 0.4 * "x");
    "acc" := "acc" + "phi";
    "x" := "feat_16";
    "phi" := "w0b_10_16" * "x" / (1.0 + EXP(-"x"));
    "phi" := "phi" + "w0c_10_16_1" * SIN(1 * 0.4 * "x") + "w0d_10_16_1" * COS(1 * 0.4 * "x");
    "phi" := "phi" + "w0c_10_16_2" * SIN(2 * 0.4 * "x") + "w0d_10_16_2" * COS(2 * 0.4 * "x");
    "phi" := "phi" + "w0c_10_16_3" * SIN(3 * 0.4 * "x") + "w0d_10_16_3" * COS(3 * 0.4 * "x");
    "phi" := "phi" + "w0c_10_16_4" * SIN(4 * 0.4 * "x") + "w0d_10_16_4" * COS(4 * 0.4 * "x");
    "phi" := "phi" + "w0c_10_16_5" * SIN(5 * 0.4 * "x") + "w0d_10_16_5" * COS(5 * 0.4 * "x");
    "phi" := "phi" + "w0c_10_16_6" * SIN(6 * 0.4 * "x") + "w0d_10_16_6" * COS(6 * 0.4 * "x");
    "acc" := "acc" + "phi";
    "x" := "feat_17";
    "phi" := "w0b_10_17" * "x" / (1.0 + EXP(-"x"));
    "phi" := "phi" + "w0c_10_17_1" * SIN(1 * 0.4 * "x") + "w0d_10_17_1" * COS(1 * 0.4 * "x");
    "phi" := "phi" + "w0c_10_17_2" * SIN(2 * 0.4 * "x") + "w0d_10_17_2" * COS(2 * 0.4 * "x");
    "phi" := "phi" + "w0c_10_17_3" * SIN(3 * 0.4 * "x") + "w0d_10_17_3" * COS(3 * 0.4 * "x");
    "phi" := "phi" + "w0c_10_17_4" * SIN(4 * 0.4 * "x") + "w0d_10_17_4" * COS(4 * 0.4 * "x");
    "phi" := "phi" + "w0c_10_17_5" * SIN(5 * 0.4 * "x") + "w0d_10_17_5" * COS(5 * 0.4 * "x");
    "phi" := "phi" + "w0c_10_17_6" * SIN(6 * 0.4 * "x") + "w0d_10_17_6" * COS(6 * 0.4 * "x");
    "acc" := "acc" + "phi";
    "x" := "feat_18";
    "phi" := "w0b_10_18" * "x" / (1.0 + EXP(-"x"));
    "phi" := "phi" + "w0c_10_18_1" * SIN(1 * 0.4 * "x") + "w0d_10_18_1" * COS(1 * 0.4 * "x");
    "phi" := "phi" + "w0c_10_18_2" * SIN(2 * 0.4 * "x") + "w0d_10_18_2" * COS(2 * 0.4 * "x");
    "phi" := "phi" + "w0c_10_18_3" * SIN(3 * 0.4 * "x") + "w0d_10_18_3" * COS(3 * 0.4 * "x");
    "phi" := "phi" + "w0c_10_18_4" * SIN(4 * 0.4 * "x") + "w0d_10_18_4" * COS(4 * 0.4 * "x");
    "phi" := "phi" + "w0c_10_18_5" * SIN(5 * 0.4 * "x") + "w0d_10_18_5" * COS(5 * 0.4 * "x");
    "phi" := "phi" + "w0c_10_18_6" * SIN(6 * 0.4 * "x") + "w0d_10_18_6" * COS(6 * 0.4 * "x");
    "acc" := "acc" + "phi";
    "x" := "feat_19";
    "phi" := "w0b_10_19" * "x" / (1.0 + EXP(-"x"));
    "phi" := "phi" + "w0c_10_19_1" * SIN(1 * 0.4 * "x") + "w0d_10_19_1" * COS(1 * 0.4 * "x");
    "phi" := "phi" + "w0c_10_19_2" * SIN(2 * 0.4 * "x") + "w0d_10_19_2" * COS(2 * 0.4 * "x");
    "phi" := "phi" + "w0c_10_19_3" * SIN(3 * 0.4 * "x") + "w0d_10_19_3" * COS(3 * 0.4 * "x");
    "phi" := "phi" + "w0c_10_19_4" * SIN(4 * 0.4 * "x") + "w0d_10_19_4" * COS(4 * 0.4 * "x");
    "phi" := "phi" + "w0c_10_19_5" * SIN(5 * 0.4 * "x") + "w0d_10_19_5" * COS(5 * 0.4 * "x");
    "phi" := "phi" + "w0c_10_19_6" * SIN(6 * 0.4 * "x") + "w0d_10_19_6" * COS(6 * 0.4 * "x");
    "acc" := "acc" + "phi";
    "x" := "feat_20";
    "phi" := "w0b_10_20" * "x" / (1.0 + EXP(-"x"));
    "phi" := "phi" + "w0c_10_20_1" * SIN(1 * 0.4 * "x") + "w0d_10_20_1" * COS(1 * 0.4 * "x");
    "phi" := "phi" + "w0c_10_20_2" * SIN(2 * 0.4 * "x") + "w0d_10_20_2" * COS(2 * 0.4 * "x");
    "phi" := "phi" + "w0c_10_20_3" * SIN(3 * 0.4 * "x") + "w0d_10_20_3" * COS(3 * 0.4 * "x");
    "phi" := "phi" + "w0c_10_20_4" * SIN(4 * 0.4 * "x") + "w0d_10_20_4" * COS(4 * 0.4 * "x");
    "phi" := "phi" + "w0c_10_20_5" * SIN(5 * 0.4 * "x") + "w0d_10_20_5" * COS(5 * 0.4 * "x");
    "phi" := "phi" + "w0c_10_20_6" * SIN(6 * 0.4 * "x") + "w0d_10_20_6" * COS(6 * 0.4 * "x");
    "acc" := "acc" + "phi";
    "x" := "feat_21";
    "phi" := "w0b_10_21" * "x" / (1.0 + EXP(-"x"));
    "phi" := "phi" + "w0c_10_21_1" * SIN(1 * 0.4 * "x") + "w0d_10_21_1" * COS(1 * 0.4 * "x");
    "phi" := "phi" + "w0c_10_21_2" * SIN(2 * 0.4 * "x") + "w0d_10_21_2" * COS(2 * 0.4 * "x");
    "phi" := "phi" + "w0c_10_21_3" * SIN(3 * 0.4 * "x") + "w0d_10_21_3" * COS(3 * 0.4 * "x");
    "phi" := "phi" + "w0c_10_21_4" * SIN(4 * 0.4 * "x") + "w0d_10_21_4" * COS(4 * 0.4 * "x");
    "phi" := "phi" + "w0c_10_21_5" * SIN(5 * 0.4 * "x") + "w0d_10_21_5" * COS(5 * 0.4 * "x");
    "phi" := "phi" + "w0c_10_21_6" * SIN(6 * 0.4 * "x") + "w0d_10_21_6" * COS(6 * 0.4 * "x");
    "acc" := "acc" + "phi";
    "x" := "feat_22";
    "phi" := "w0b_10_22" * "x" / (1.0 + EXP(-"x"));
    "phi" := "phi" + "w0c_10_22_1" * SIN(1 * 0.4 * "x") + "w0d_10_22_1" * COS(1 * 0.4 * "x");
    "phi" := "phi" + "w0c_10_22_2" * SIN(2 * 0.4 * "x") + "w0d_10_22_2" * COS(2 * 0.4 * "x");
    "phi" := "phi" + "w0c_10_22_3" * SIN(3 * 0.4 * "x") + "w0d_10_22_3" * COS(3 * 0.4 * "x");
    "phi" := "phi" + "w0c_10_22_4" * SIN(4 * 0.4 * "x") + "w0d_10_22_4" * COS(4 * 0.4 * "x");
    "phi" := "phi" + "w0c_10_22_5" * SIN(5 * 0.4 * "x") + "w0d_10_22_5" * COS(5 * 0.4 * "x");
    "phi" := "phi" + "w0c_10_22_6" * SIN(6 * 0.4 * "x") + "w0d_10_22_6" * COS(6 * 0.4 * "x");
    "acc" := "acc" + "phi";
    "x" := "feat_23";
    "phi" := "w0b_10_23" * "x" / (1.0 + EXP(-"x"));
    "phi" := "phi" + "w0c_10_23_1" * SIN(1 * 0.4 * "x") + "w0d_10_23_1" * COS(1 * 0.4 * "x");
    "phi" := "phi" + "w0c_10_23_2" * SIN(2 * 0.4 * "x") + "w0d_10_23_2" * COS(2 * 0.4 * "x");
    "phi" := "phi" + "w0c_10_23_3" * SIN(3 * 0.4 * "x") + "w0d_10_23_3" * COS(3 * 0.4 * "x");
    "phi" := "phi" + "w0c_10_23_4" * SIN(4 * 0.4 * "x") + "w0d_10_23_4" * COS(4 * 0.4 * "x");
    "phi" := "phi" + "w0c_10_23_5" * SIN(5 * 0.4 * "x") + "w0d_10_23_5" * COS(5 * 0.4 * "x");
    "phi" := "phi" + "w0c_10_23_6" * SIN(6 * 0.4 * "x") + "w0d_10_23_6" * COS(6 * 0.4 * "x");
    "acc" := "acc" + "phi";
    "x" := "feat_24";
    "phi" := "w0b_10_24" * "x" / (1.0 + EXP(-"x"));
    "phi" := "phi" + "w0c_10_24_1" * SIN(1 * 0.4 * "x") + "w0d_10_24_1" * COS(1 * 0.4 * "x");
    "phi" := "phi" + "w0c_10_24_2" * SIN(2 * 0.4 * "x") + "w0d_10_24_2" * COS(2 * 0.4 * "x");
    "phi" := "phi" + "w0c_10_24_3" * SIN(3 * 0.4 * "x") + "w0d_10_24_3" * COS(3 * 0.4 * "x");
    "phi" := "phi" + "w0c_10_24_4" * SIN(4 * 0.4 * "x") + "w0d_10_24_4" * COS(4 * 0.4 * "x");
    "phi" := "phi" + "w0c_10_24_5" * SIN(5 * 0.4 * "x") + "w0d_10_24_5" * COS(5 * 0.4 * "x");
    "phi" := "phi" + "w0c_10_24_6" * SIN(6 * 0.4 * "x") + "w0d_10_24_6" * COS(6 * 0.4 * "x");
    "acc" := "acc" + "phi";
    "x" := "feat_25";
    "phi" := "w0b_10_25" * "x" / (1.0 + EXP(-"x"));
    "phi" := "phi" + "w0c_10_25_1" * SIN(1 * 0.4 * "x") + "w0d_10_25_1" * COS(1 * 0.4 * "x");
    "phi" := "phi" + "w0c_10_25_2" * SIN(2 * 0.4 * "x") + "w0d_10_25_2" * COS(2 * 0.4 * "x");
    "phi" := "phi" + "w0c_10_25_3" * SIN(3 * 0.4 * "x") + "w0d_10_25_3" * COS(3 * 0.4 * "x");
    "phi" := "phi" + "w0c_10_25_4" * SIN(4 * 0.4 * "x") + "w0d_10_25_4" * COS(4 * 0.4 * "x");
    "phi" := "phi" + "w0c_10_25_5" * SIN(5 * 0.4 * "x") + "w0d_10_25_5" * COS(5 * 0.4 * "x");
    "phi" := "phi" + "w0c_10_25_6" * SIN(6 * 0.4 * "x") + "w0d_10_25_6" * COS(6 * 0.4 * "x");
    "acc" := "acc" + "phi";
    "x" := "feat_26";
    "phi" := "w0b_10_26" * "x" / (1.0 + EXP(-"x"));
    "phi" := "phi" + "w0c_10_26_1" * SIN(1 * 0.4 * "x") + "w0d_10_26_1" * COS(1 * 0.4 * "x");
    "phi" := "phi" + "w0c_10_26_2" * SIN(2 * 0.4 * "x") + "w0d_10_26_2" * COS(2 * 0.4 * "x");
    "phi" := "phi" + "w0c_10_26_3" * SIN(3 * 0.4 * "x") + "w0d_10_26_3" * COS(3 * 0.4 * "x");
    "phi" := "phi" + "w0c_10_26_4" * SIN(4 * 0.4 * "x") + "w0d_10_26_4" * COS(4 * 0.4 * "x");
    "phi" := "phi" + "w0c_10_26_5" * SIN(5 * 0.4 * "x") + "w0d_10_26_5" * COS(5 * 0.4 * "x");
    "phi" := "phi" + "w0c_10_26_6" * SIN(6 * 0.4 * "x") + "w0d_10_26_6" * COS(6 * 0.4 * "x");
    "acc" := "acc" + "phi";
    "x" := "feat_27";
    "phi" := "w0b_10_27" * "x" / (1.0 + EXP(-"x"));
    "phi" := "phi" + "w0c_10_27_1" * SIN(1 * 0.4 * "x") + "w0d_10_27_1" * COS(1 * 0.4 * "x");
    "phi" := "phi" + "w0c_10_27_2" * SIN(2 * 0.4 * "x") + "w0d_10_27_2" * COS(2 * 0.4 * "x");
    "phi" := "phi" + "w0c_10_27_3" * SIN(3 * 0.4 * "x") + "w0d_10_27_3" * COS(3 * 0.4 * "x");
    "phi" := "phi" + "w0c_10_27_4" * SIN(4 * 0.4 * "x") + "w0d_10_27_4" * COS(4 * 0.4 * "x");
    "phi" := "phi" + "w0c_10_27_5" * SIN(5 * 0.4 * "x") + "w0d_10_27_5" * COS(5 * 0.4 * "x");
    "phi" := "phi" + "w0c_10_27_6" * SIN(6 * 0.4 * "x") + "w0d_10_27_6" * COS(6 * 0.4 * "x");
    "acc" := "acc" + "phi";
    "x" := "feat_28";
    "phi" := "w0b_10_28" * "x" / (1.0 + EXP(-"x"));
    "phi" := "phi" + "w0c_10_28_1" * SIN(1 * 0.4 * "x") + "w0d_10_28_1" * COS(1 * 0.4 * "x");
    "phi" := "phi" + "w0c_10_28_2" * SIN(2 * 0.4 * "x") + "w0d_10_28_2" * COS(2 * 0.4 * "x");
    "phi" := "phi" + "w0c_10_28_3" * SIN(3 * 0.4 * "x") + "w0d_10_28_3" * COS(3 * 0.4 * "x");
    "phi" := "phi" + "w0c_10_28_4" * SIN(4 * 0.4 * "x") + "w0d_10_28_4" * COS(4 * 0.4 * "x");
    "phi" := "phi" + "w0c_10_28_5" * SIN(5 * 0.4 * "x") + "w0d_10_28_5" * COS(5 * 0.4 * "x");
    "phi" := "phi" + "w0c_10_28_6" * SIN(6 * 0.4 * "x") + "w0d_10_28_6" * COS(6 * 0.4 * "x");
    "acc" := "acc" + "phi";
    "h1_10" := "acc" + "b0_10";
    "acc" := 0.0;
    "x" := "feat_1";
    "phi" := "w0b_11_1" * "x" / (1.0 + EXP(-"x"));
    "phi" := "phi" + "w0c_11_1_1" * SIN(1 * 0.4 * "x") + "w0d_11_1_1" * COS(1 * 0.4 * "x");
    "phi" := "phi" + "w0c_11_1_2" * SIN(2 * 0.4 * "x") + "w0d_11_1_2" * COS(2 * 0.4 * "x");
    "phi" := "phi" + "w0c_11_1_3" * SIN(3 * 0.4 * "x") + "w0d_11_1_3" * COS(3 * 0.4 * "x");
    "phi" := "phi" + "w0c_11_1_4" * SIN(4 * 0.4 * "x") + "w0d_11_1_4" * COS(4 * 0.4 * "x");
    "phi" := "phi" + "w0c_11_1_5" * SIN(5 * 0.4 * "x") + "w0d_11_1_5" * COS(5 * 0.4 * "x");
    "phi" := "phi" + "w0c_11_1_6" * SIN(6 * 0.4 * "x") + "w0d_11_1_6" * COS(6 * 0.4 * "x");
    "acc" := "acc" + "phi";
    "x" := "feat_2";
    "phi" := "w0b_11_2" * "x" / (1.0 + EXP(-"x"));
    "phi" := "phi" + "w0c_11_2_1" * SIN(1 * 0.4 * "x") + "w0d_11_2_1" * COS(1 * 0.4 * "x");
    "phi" := "phi" + "w0c_11_2_2" * SIN(2 * 0.4 * "x") + "w0d_11_2_2" * COS(2 * 0.4 * "x");
    "phi" := "phi" + "w0c_11_2_3" * SIN(3 * 0.4 * "x") + "w0d_11_2_3" * COS(3 * 0.4 * "x");
    "phi" := "phi" + "w0c_11_2_4" * SIN(4 * 0.4 * "x") + "w0d_11_2_4" * COS(4 * 0.4 * "x");
    "phi" := "phi" + "w0c_11_2_5" * SIN(5 * 0.4 * "x") + "w0d_11_2_5" * COS(5 * 0.4 * "x");
    "phi" := "phi" + "w0c_11_2_6" * SIN(6 * 0.4 * "x") + "w0d_11_2_6" * COS(6 * 0.4 * "x");
    "acc" := "acc" + "phi";
    "x" := "feat_3";
    "phi" := "w0b_11_3" * "x" / (1.0 + EXP(-"x"));
    "phi" := "phi" + "w0c_11_3_1" * SIN(1 * 0.4 * "x") + "w0d_11_3_1" * COS(1 * 0.4 * "x");
    "phi" := "phi" + "w0c_11_3_2" * SIN(2 * 0.4 * "x") + "w0d_11_3_2" * COS(2 * 0.4 * "x");
    "phi" := "phi" + "w0c_11_3_3" * SIN(3 * 0.4 * "x") + "w0d_11_3_3" * COS(3 * 0.4 * "x");
    "phi" := "phi" + "w0c_11_3_4" * SIN(4 * 0.4 * "x") + "w0d_11_3_4" * COS(4 * 0.4 * "x");
    "phi" := "phi" + "w0c_11_3_5" * SIN(5 * 0.4 * "x") + "w0d_11_3_5" * COS(5 * 0.4 * "x");
    "phi" := "phi" + "w0c_11_3_6" * SIN(6 * 0.4 * "x") + "w0d_11_3_6" * COS(6 * 0.4 * "x");
    "acc" := "acc" + "phi";
    "x" := "feat_4";
    "phi" := "w0b_11_4" * "x" / (1.0 + EXP(-"x"));
    "phi" := "phi" + "w0c_11_4_1" * SIN(1 * 0.4 * "x") + "w0d_11_4_1" * COS(1 * 0.4 * "x");
    "phi" := "phi" + "w0c_11_4_2" * SIN(2 * 0.4 * "x") + "w0d_11_4_2" * COS(2 * 0.4 * "x");
    "phi" := "phi" + "w0c_11_4_3" * SIN(3 * 0.4 * "x") + "w0d_11_4_3" * COS(3 * 0.4 * "x");
    "phi" := "phi" + "w0c_11_4_4" * SIN(4 * 0.4 * "x") + "w0d_11_4_4" * COS(4 * 0.4 * "x");
    "phi" := "phi" + "w0c_11_4_5" * SIN(5 * 0.4 * "x") + "w0d_11_4_5" * COS(5 * 0.4 * "x");
    "phi" := "phi" + "w0c_11_4_6" * SIN(6 * 0.4 * "x") + "w0d_11_4_6" * COS(6 * 0.4 * "x");
    "acc" := "acc" + "phi";
    "x" := "feat_5";
    "phi" := "w0b_11_5" * "x" / (1.0 + EXP(-"x"));
    "phi" := "phi" + "w0c_11_5_1" * SIN(1 * 0.4 * "x") + "w0d_11_5_1" * COS(1 * 0.4 * "x");
    "phi" := "phi" + "w0c_11_5_2" * SIN(2 * 0.4 * "x") + "w0d_11_5_2" * COS(2 * 0.4 * "x");
    "phi" := "phi" + "w0c_11_5_3" * SIN(3 * 0.4 * "x") + "w0d_11_5_3" * COS(3 * 0.4 * "x");
    "phi" := "phi" + "w0c_11_5_4" * SIN(4 * 0.4 * "x") + "w0d_11_5_4" * COS(4 * 0.4 * "x");
    "phi" := "phi" + "w0c_11_5_5" * SIN(5 * 0.4 * "x") + "w0d_11_5_5" * COS(5 * 0.4 * "x");
    "phi" := "phi" + "w0c_11_5_6" * SIN(6 * 0.4 * "x") + "w0d_11_5_6" * COS(6 * 0.4 * "x");
    "acc" := "acc" + "phi";
    "x" := "feat_6";
    "phi" := "w0b_11_6" * "x" / (1.0 + EXP(-"x"));
    "phi" := "phi" + "w0c_11_6_1" * SIN(1 * 0.4 * "x") + "w0d_11_6_1" * COS(1 * 0.4 * "x");
    "phi" := "phi" + "w0c_11_6_2" * SIN(2 * 0.4 * "x") + "w0d_11_6_2" * COS(2 * 0.4 * "x");
    "phi" := "phi" + "w0c_11_6_3" * SIN(3 * 0.4 * "x") + "w0d_11_6_3" * COS(3 * 0.4 * "x");
    "phi" := "phi" + "w0c_11_6_4" * SIN(4 * 0.4 * "x") + "w0d_11_6_4" * COS(4 * 0.4 * "x");
    "phi" := "phi" + "w0c_11_6_5" * SIN(5 * 0.4 * "x") + "w0d_11_6_5" * COS(5 * 0.4 * "x");
    "phi" := "phi" + "w0c_11_6_6" * SIN(6 * 0.4 * "x") + "w0d_11_6_6" * COS(6 * 0.4 * "x");
    "acc" := "acc" + "phi";
    "x" := "feat_7";
    "phi" := "w0b_11_7" * "x" / (1.0 + EXP(-"x"));
    "phi" := "phi" + "w0c_11_7_1" * SIN(1 * 0.4 * "x") + "w0d_11_7_1" * COS(1 * 0.4 * "x");
    "phi" := "phi" + "w0c_11_7_2" * SIN(2 * 0.4 * "x") + "w0d_11_7_2" * COS(2 * 0.4 * "x");
    "phi" := "phi" + "w0c_11_7_3" * SIN(3 * 0.4 * "x") + "w0d_11_7_3" * COS(3 * 0.4 * "x");
    "phi" := "phi" + "w0c_11_7_4" * SIN(4 * 0.4 * "x") + "w0d_11_7_4" * COS(4 * 0.4 * "x");
    "phi" := "phi" + "w0c_11_7_5" * SIN(5 * 0.4 * "x") + "w0d_11_7_5" * COS(5 * 0.4 * "x");
    "phi" := "phi" + "w0c_11_7_6" * SIN(6 * 0.4 * "x") + "w0d_11_7_6" * COS(6 * 0.4 * "x");
    "acc" := "acc" + "phi";
    "x" := "feat_8";
    "phi" := "w0b_11_8" * "x" / (1.0 + EXP(-"x"));
    "phi" := "phi" + "w0c_11_8_1" * SIN(1 * 0.4 * "x") + "w0d_11_8_1" * COS(1 * 0.4 * "x");
    "phi" := "phi" + "w0c_11_8_2" * SIN(2 * 0.4 * "x") + "w0d_11_8_2" * COS(2 * 0.4 * "x");
    "phi" := "phi" + "w0c_11_8_3" * SIN(3 * 0.4 * "x") + "w0d_11_8_3" * COS(3 * 0.4 * "x");
    "phi" := "phi" + "w0c_11_8_4" * SIN(4 * 0.4 * "x") + "w0d_11_8_4" * COS(4 * 0.4 * "x");
    "phi" := "phi" + "w0c_11_8_5" * SIN(5 * 0.4 * "x") + "w0d_11_8_5" * COS(5 * 0.4 * "x");
    "phi" := "phi" + "w0c_11_8_6" * SIN(6 * 0.4 * "x") + "w0d_11_8_6" * COS(6 * 0.4 * "x");
    "acc" := "acc" + "phi";
    "x" := "feat_9";
    "phi" := "w0b_11_9" * "x" / (1.0 + EXP(-"x"));
    "phi" := "phi" + "w0c_11_9_1" * SIN(1 * 0.4 * "x") + "w0d_11_9_1" * COS(1 * 0.4 * "x");
    "phi" := "phi" + "w0c_11_9_2" * SIN(2 * 0.4 * "x") + "w0d_11_9_2" * COS(2 * 0.4 * "x");
    "phi" := "phi" + "w0c_11_9_3" * SIN(3 * 0.4 * "x") + "w0d_11_9_3" * COS(3 * 0.4 * "x");
    "phi" := "phi" + "w0c_11_9_4" * SIN(4 * 0.4 * "x") + "w0d_11_9_4" * COS(4 * 0.4 * "x");
    "phi" := "phi" + "w0c_11_9_5" * SIN(5 * 0.4 * "x") + "w0d_11_9_5" * COS(5 * 0.4 * "x");
    "phi" := "phi" + "w0c_11_9_6" * SIN(6 * 0.4 * "x") + "w0d_11_9_6" * COS(6 * 0.4 * "x");
    "acc" := "acc" + "phi";
    "x" := "feat_10";
    "phi" := "w0b_11_10" * "x" / (1.0 + EXP(-"x"));
    "phi" := "phi" + "w0c_11_10_1" * SIN(1 * 0.4 * "x") + "w0d_11_10_1" * COS(1 * 0.4 * "x");
    "phi" := "phi" + "w0c_11_10_2" * SIN(2 * 0.4 * "x") + "w0d_11_10_2" * COS(2 * 0.4 * "x");
    "phi" := "phi" + "w0c_11_10_3" * SIN(3 * 0.4 * "x") + "w0d_11_10_3" * COS(3 * 0.4 * "x");
    "phi" := "phi" + "w0c_11_10_4" * SIN(4 * 0.4 * "x") + "w0d_11_10_4" * COS(4 * 0.4 * "x");
    "phi" := "phi" + "w0c_11_10_5" * SIN(5 * 0.4 * "x") + "w0d_11_10_5" * COS(5 * 0.4 * "x");
    "phi" := "phi" + "w0c_11_10_6" * SIN(6 * 0.4 * "x") + "w0d_11_10_6" * COS(6 * 0.4 * "x");
    "acc" := "acc" + "phi";
    "x" := "feat_11";
    "phi" := "w0b_11_11" * "x" / (1.0 + EXP(-"x"));
    "phi" := "phi" + "w0c_11_11_1" * SIN(1 * 0.4 * "x") + "w0d_11_11_1" * COS(1 * 0.4 * "x");
    "phi" := "phi" + "w0c_11_11_2" * SIN(2 * 0.4 * "x") + "w0d_11_11_2" * COS(2 * 0.4 * "x");
    "phi" := "phi" + "w0c_11_11_3" * SIN(3 * 0.4 * "x") + "w0d_11_11_3" * COS(3 * 0.4 * "x");
    "phi" := "phi" + "w0c_11_11_4" * SIN(4 * 0.4 * "x") + "w0d_11_11_4" * COS(4 * 0.4 * "x");
    "phi" := "phi" + "w0c_11_11_5" * SIN(5 * 0.4 * "x") + "w0d_11_11_5" * COS(5 * 0.4 * "x");
    "phi" := "phi" + "w0c_11_11_6" * SIN(6 * 0.4 * "x") + "w0d_11_11_6" * COS(6 * 0.4 * "x");
    "acc" := "acc" + "phi";
    "x" := "feat_12";
    "phi" := "w0b_11_12" * "x" / (1.0 + EXP(-"x"));
    "phi" := "phi" + "w0c_11_12_1" * SIN(1 * 0.4 * "x") + "w0d_11_12_1" * COS(1 * 0.4 * "x");
    "phi" := "phi" + "w0c_11_12_2" * SIN(2 * 0.4 * "x") + "w0d_11_12_2" * COS(2 * 0.4 * "x");
    "phi" := "phi" + "w0c_11_12_3" * SIN(3 * 0.4 * "x") + "w0d_11_12_3" * COS(3 * 0.4 * "x");
    "phi" := "phi" + "w0c_11_12_4" * SIN(4 * 0.4 * "x") + "w0d_11_12_4" * COS(4 * 0.4 * "x");
    "phi" := "phi" + "w0c_11_12_5" * SIN(5 * 0.4 * "x") + "w0d_11_12_5" * COS(5 * 0.4 * "x");
    "phi" := "phi" + "w0c_11_12_6" * SIN(6 * 0.4 * "x") + "w0d_11_12_6" * COS(6 * 0.4 * "x");
    "acc" := "acc" + "phi";
    "x" := "feat_13";
    "phi" := "w0b_11_13" * "x" / (1.0 + EXP(-"x"));
    "phi" := "phi" + "w0c_11_13_1" * SIN(1 * 0.4 * "x") + "w0d_11_13_1" * COS(1 * 0.4 * "x");
    "phi" := "phi" + "w0c_11_13_2" * SIN(2 * 0.4 * "x") + "w0d_11_13_2" * COS(2 * 0.4 * "x");
    "phi" := "phi" + "w0c_11_13_3" * SIN(3 * 0.4 * "x") + "w0d_11_13_3" * COS(3 * 0.4 * "x");
    "phi" := "phi" + "w0c_11_13_4" * SIN(4 * 0.4 * "x") + "w0d_11_13_4" * COS(4 * 0.4 * "x");
    "phi" := "phi" + "w0c_11_13_5" * SIN(5 * 0.4 * "x") + "w0d_11_13_5" * COS(5 * 0.4 * "x");
    "phi" := "phi" + "w0c_11_13_6" * SIN(6 * 0.4 * "x") + "w0d_11_13_6" * COS(6 * 0.4 * "x");
    "acc" := "acc" + "phi";
    "x" := "feat_14";
    "phi" := "w0b_11_14" * "x" / (1.0 + EXP(-"x"));
    "phi" := "phi" + "w0c_11_14_1" * SIN(1 * 0.4 * "x") + "w0d_11_14_1" * COS(1 * 0.4 * "x");
    "phi" := "phi" + "w0c_11_14_2" * SIN(2 * 0.4 * "x") + "w0d_11_14_2" * COS(2 * 0.4 * "x");
    "phi" := "phi" + "w0c_11_14_3" * SIN(3 * 0.4 * "x") + "w0d_11_14_3" * COS(3 * 0.4 * "x");
    "phi" := "phi" + "w0c_11_14_4" * SIN(4 * 0.4 * "x") + "w0d_11_14_4" * COS(4 * 0.4 * "x");
    "phi" := "phi" + "w0c_11_14_5" * SIN(5 * 0.4 * "x") + "w0d_11_14_5" * COS(5 * 0.4 * "x");
    "phi" := "phi" + "w0c_11_14_6" * SIN(6 * 0.4 * "x") + "w0d_11_14_6" * COS(6 * 0.4 * "x");
    "acc" := "acc" + "phi";
    "x" := "feat_15";
    "phi" := "w0b_11_15" * "x" / (1.0 + EXP(-"x"));
    "phi" := "phi" + "w0c_11_15_1" * SIN(1 * 0.4 * "x") + "w0d_11_15_1" * COS(1 * 0.4 * "x");
    "phi" := "phi" + "w0c_11_15_2" * SIN(2 * 0.4 * "x") + "w0d_11_15_2" * COS(2 * 0.4 * "x");
    "phi" := "phi" + "w0c_11_15_3" * SIN(3 * 0.4 * "x") + "w0d_11_15_3" * COS(3 * 0.4 * "x");
    "phi" := "phi" + "w0c_11_15_4" * SIN(4 * 0.4 * "x") + "w0d_11_15_4" * COS(4 * 0.4 * "x");
    "phi" := "phi" + "w0c_11_15_5" * SIN(5 * 0.4 * "x") + "w0d_11_15_5" * COS(5 * 0.4 * "x");
    "phi" := "phi" + "w0c_11_15_6" * SIN(6 * 0.4 * "x") + "w0d_11_15_6" * COS(6 * 0.4 * "x");
    "acc" := "acc" + "phi";
    "x" := "feat_16";
    "phi" := "w0b_11_16" * "x" / (1.0 + EXP(-"x"));
    "phi" := "phi" + "w0c_11_16_1" * SIN(1 * 0.4 * "x") + "w0d_11_16_1" * COS(1 * 0.4 * "x");
    "phi" := "phi" + "w0c_11_16_2" * SIN(2 * 0.4 * "x") + "w0d_11_16_2" * COS(2 * 0.4 * "x");
    "phi" := "phi" + "w0c_11_16_3" * SIN(3 * 0.4 * "x") + "w0d_11_16_3" * COS(3 * 0.4 * "x");
    "phi" := "phi" + "w0c_11_16_4" * SIN(4 * 0.4 * "x") + "w0d_11_16_4" * COS(4 * 0.4 * "x");
    "phi" := "phi" + "w0c_11_16_5" * SIN(5 * 0.4 * "x") + "w0d_11_16_5" * COS(5 * 0.4 * "x");
    "phi" := "phi" + "w0c_11_16_6" * SIN(6 * 0.4 * "x") + "w0d_11_16_6" * COS(6 * 0.4 * "x");
    "acc" := "acc" + "phi";
    "x" := "feat_17";
    "phi" := "w0b_11_17" * "x" / (1.0 + EXP(-"x"));
    "phi" := "phi" + "w0c_11_17_1" * SIN(1 * 0.4 * "x") + "w0d_11_17_1" * COS(1 * 0.4 * "x");
    "phi" := "phi" + "w0c_11_17_2" * SIN(2 * 0.4 * "x") + "w0d_11_17_2" * COS(2 * 0.4 * "x");
    "phi" := "phi" + "w0c_11_17_3" * SIN(3 * 0.4 * "x") + "w0d_11_17_3" * COS(3 * 0.4 * "x");
    "phi" := "phi" + "w0c_11_17_4" * SIN(4 * 0.4 * "x") + "w0d_11_17_4" * COS(4 * 0.4 * "x");
    "phi" := "phi" + "w0c_11_17_5" * SIN(5 * 0.4 * "x") + "w0d_11_17_5" * COS(5 * 0.4 * "x");
    "phi" := "phi" + "w0c_11_17_6" * SIN(6 * 0.4 * "x") + "w0d_11_17_6" * COS(6 * 0.4 * "x");
    "acc" := "acc" + "phi";
    "x" := "feat_18";
    "phi" := "w0b_11_18" * "x" / (1.0 + EXP(-"x"));
    "phi" := "phi" + "w0c_11_18_1" * SIN(1 * 0.4 * "x") + "w0d_11_18_1" * COS(1 * 0.4 * "x");
    "phi" := "phi" + "w0c_11_18_2" * SIN(2 * 0.4 * "x") + "w0d_11_18_2" * COS(2 * 0.4 * "x");
    "phi" := "phi" + "w0c_11_18_3" * SIN(3 * 0.4 * "x") + "w0d_11_18_3" * COS(3 * 0.4 * "x");
    "phi" := "phi" + "w0c_11_18_4" * SIN(4 * 0.4 * "x") + "w0d_11_18_4" * COS(4 * 0.4 * "x");
    "phi" := "phi" + "w0c_11_18_5" * SIN(5 * 0.4 * "x") + "w0d_11_18_5" * COS(5 * 0.4 * "x");
    "phi" := "phi" + "w0c_11_18_6" * SIN(6 * 0.4 * "x") + "w0d_11_18_6" * COS(6 * 0.4 * "x");
    "acc" := "acc" + "phi";
    "x" := "feat_19";
    "phi" := "w0b_11_19" * "x" / (1.0 + EXP(-"x"));
    "phi" := "phi" + "w0c_11_19_1" * SIN(1 * 0.4 * "x") + "w0d_11_19_1" * COS(1 * 0.4 * "x");
    "phi" := "phi" + "w0c_11_19_2" * SIN(2 * 0.4 * "x") + "w0d_11_19_2" * COS(2 * 0.4 * "x");
    "phi" := "phi" + "w0c_11_19_3" * SIN(3 * 0.4 * "x") + "w0d_11_19_3" * COS(3 * 0.4 * "x");
    "phi" := "phi" + "w0c_11_19_4" * SIN(4 * 0.4 * "x") + "w0d_11_19_4" * COS(4 * 0.4 * "x");
    "phi" := "phi" + "w0c_11_19_5" * SIN(5 * 0.4 * "x") + "w0d_11_19_5" * COS(5 * 0.4 * "x");
    "phi" := "phi" + "w0c_11_19_6" * SIN(6 * 0.4 * "x") + "w0d_11_19_6" * COS(6 * 0.4 * "x");
    "acc" := "acc" + "phi";
    "x" := "feat_20";
    "phi" := "w0b_11_20" * "x" / (1.0 + EXP(-"x"));
    "phi" := "phi" + "w0c_11_20_1" * SIN(1 * 0.4 * "x") + "w0d_11_20_1" * COS(1 * 0.4 * "x");
    "phi" := "phi" + "w0c_11_20_2" * SIN(2 * 0.4 * "x") + "w0d_11_20_2" * COS(2 * 0.4 * "x");
    "phi" := "phi" + "w0c_11_20_3" * SIN(3 * 0.4 * "x") + "w0d_11_20_3" * COS(3 * 0.4 * "x");
    "phi" := "phi" + "w0c_11_20_4" * SIN(4 * 0.4 * "x") + "w0d_11_20_4" * COS(4 * 0.4 * "x");
    "phi" := "phi" + "w0c_11_20_5" * SIN(5 * 0.4 * "x") + "w0d_11_20_5" * COS(5 * 0.4 * "x");
    "phi" := "phi" + "w0c_11_20_6" * SIN(6 * 0.4 * "x") + "w0d_11_20_6" * COS(6 * 0.4 * "x");
    "acc" := "acc" + "phi";
    "x" := "feat_21";
    "phi" := "w0b_11_21" * "x" / (1.0 + EXP(-"x"));
    "phi" := "phi" + "w0c_11_21_1" * SIN(1 * 0.4 * "x") + "w0d_11_21_1" * COS(1 * 0.4 * "x");
    "phi" := "phi" + "w0c_11_21_2" * SIN(2 * 0.4 * "x") + "w0d_11_21_2" * COS(2 * 0.4 * "x");
    "phi" := "phi" + "w0c_11_21_3" * SIN(3 * 0.4 * "x") + "w0d_11_21_3" * COS(3 * 0.4 * "x");
    "phi" := "phi" + "w0c_11_21_4" * SIN(4 * 0.4 * "x") + "w0d_11_21_4" * COS(4 * 0.4 * "x");
    "phi" := "phi" + "w0c_11_21_5" * SIN(5 * 0.4 * "x") + "w0d_11_21_5" * COS(5 * 0.4 * "x");
    "phi" := "phi" + "w0c_11_21_6" * SIN(6 * 0.4 * "x") + "w0d_11_21_6" * COS(6 * 0.4 * "x");
    "acc" := "acc" + "phi";
    "x" := "feat_22";
    "phi" := "w0b_11_22" * "x" / (1.0 + EXP(-"x"));
    "phi" := "phi" + "w0c_11_22_1" * SIN(1 * 0.4 * "x") + "w0d_11_22_1" * COS(1 * 0.4 * "x");
    "phi" := "phi" + "w0c_11_22_2" * SIN(2 * 0.4 * "x") + "w0d_11_22_2" * COS(2 * 0.4 * "x");
    "phi" := "phi" + "w0c_11_22_3" * SIN(3 * 0.4 * "x") + "w0d_11_22_3" * COS(3 * 0.4 * "x");
    "phi" := "phi" + "w0c_11_22_4" * SIN(4 * 0.4 * "x") + "w0d_11_22_4" * COS(4 * 0.4 * "x");
    "phi" := "phi" + "w0c_11_22_5" * SIN(5 * 0.4 * "x") + "w0d_11_22_5" * COS(5 * 0.4 * "x");
    "phi" := "phi" + "w0c_11_22_6" * SIN(6 * 0.4 * "x") + "w0d_11_22_6" * COS(6 * 0.4 * "x");
    "acc" := "acc" + "phi";
    "x" := "feat_23";
    "phi" := "w0b_11_23" * "x" / (1.0 + EXP(-"x"));
    "phi" := "phi" + "w0c_11_23_1" * SIN(1 * 0.4 * "x") + "w0d_11_23_1" * COS(1 * 0.4 * "x");
    "phi" := "phi" + "w0c_11_23_2" * SIN(2 * 0.4 * "x") + "w0d_11_23_2" * COS(2 * 0.4 * "x");
    "phi" := "phi" + "w0c_11_23_3" * SIN(3 * 0.4 * "x") + "w0d_11_23_3" * COS(3 * 0.4 * "x");
    "phi" := "phi" + "w0c_11_23_4" * SIN(4 * 0.4 * "x") + "w0d_11_23_4" * COS(4 * 0.4 * "x");
    "phi" := "phi" + "w0c_11_23_5" * SIN(5 * 0.4 * "x") + "w0d_11_23_5" * COS(5 * 0.4 * "x");
    "phi" := "phi" + "w0c_11_23_6" * SIN(6 * 0.4 * "x") + "w0d_11_23_6" * COS(6 * 0.4 * "x");
    "acc" := "acc" + "phi";
    "x" := "feat_24";
    "phi" := "w0b_11_24" * "x" / (1.0 + EXP(-"x"));
    "phi" := "phi" + "w0c_11_24_1" * SIN(1 * 0.4 * "x") + "w0d_11_24_1" * COS(1 * 0.4 * "x");
    "phi" := "phi" + "w0c_11_24_2" * SIN(2 * 0.4 * "x") + "w0d_11_24_2" * COS(2 * 0.4 * "x");
    "phi" := "phi" + "w0c_11_24_3" * SIN(3 * 0.4 * "x") + "w0d_11_24_3" * COS(3 * 0.4 * "x");
    "phi" := "phi" + "w0c_11_24_4" * SIN(4 * 0.4 * "x") + "w0d_11_24_4" * COS(4 * 0.4 * "x");
